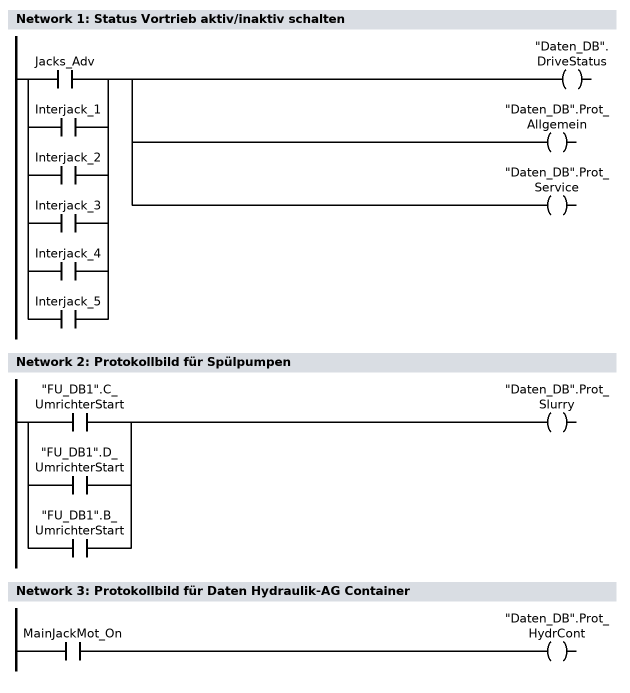
NETWORK
TITLE = Status Vortrieb aktiv/inaktiv schalten
      O     "Jacks_Adv";
      O     "Interjack_1";
      O     "Interjack_2";
      O     "Interjack_3";
      O     "Interjack_4";
      O     "Interjack_5";
      =     "Daten_DB".DriveStatus;
      =     "Daten_DB".Prot_Allgemein;
      =     "Daten_DB".Prot_Service;
NETWORK
TITLE = Protokollbild für Spülpumpen
      O     "FU_DB1".C_UmrichterStart;
      O     "FU_DB1".D_UmrichterStart;
      O     "FU_DB1".B_UmrichterStart;
      =     "Daten_DB".Prot_Slurry;
NETWORK
TITLE = Protokollbild für Daten Hydraulik-AG Container
      A     "MainJackMot_On";
      =     "Daten_DB".Prot_HydrCont;
END_FUNCTION

FUNCTION "DP Ausfall" : VOID	// FC 76
TITLE = Auswertung der Slave-Diagnose
AUTHOR : Simdon
FAMILY : Check
NAME : DP_Fail
VERSION : 0.1
BEGIN
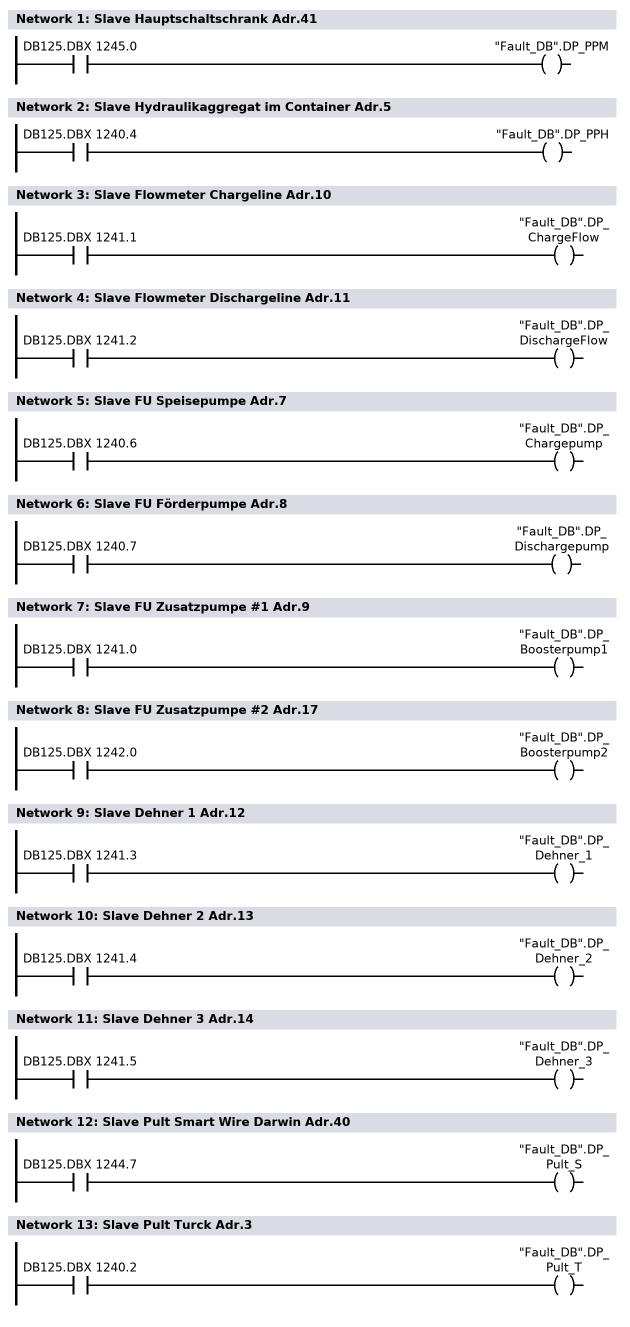
NETWORK
TITLE = Slave Hauptschaltschrank Adr.41
      A     DB125.DBX 1245.0;
      =     "Fault_DB".DP_PPM;
NETWORK
TITLE = Slave Hydraulikaggregat im Container Adr.5
      A     DB125.DBX 1240.4;
      =     "Fault_DB".DP_PPH;
NETWORK
TITLE = Slave Flowmeter Chargeline Adr.10
      A     DB125.DBX 1241.1;
      =     "Fault_DB".DP_ChargeFlow;
NETWORK
TITLE = Slave Flowmeter Dischargeline Adr.11
      A     DB125.DBX 1241.2;
      =     "Fault_DB".DP_DischargeFlow;
NETWORK
TITLE = Slave FU Speisepumpe Adr.7
      A     DB125.DBX 1240.6;
      =     "Fault_DB".DP_Chargepump;
NETWORK
TITLE = Slave FU Förderpumpe Adr.8
      A     DB125.DBX 1240.7;
      =     "Fault_DB".DP_Dischargepump;
NETWORK
TITLE = Slave FU Zusatzpumpe #1 Adr.9
      A     DB125.DBX 1241.0;
      =     "Fault_DB".DP_Boosterpump1;
NETWORK
TITLE = Slave FU Zusatzpumpe #2 Adr.17
      A     DB125.DBX 1242.0;
      =     "Fault_DB".DP_Boosterpump2;
NETWORK
TITLE = Slave Dehner 1 Adr.12
      A     DB125.DBX 1241.3;
      =     "Fault_DB".DP_Dehner_1;
NETWORK
TITLE = Slave Dehner 2 Adr.13
      A     DB125.DBX 1241.4;
      =     "Fault_DB".DP_Dehner_2;
NETWORK
TITLE = Slave Dehner 3 Adr.14
      A     DB125.DBX 1241.5;
      =     "Fault_DB".DP_Dehner_3;
NETWORK
TITLE = Slave Pult Smart Wire Darwin Adr.40
      A     DB125.DBX 1244.7;
      =     "Fault_DB".DP_Pult_S;
NETWORK
TITLE = Slave Pult Turck Adr.3
      A     DB125.DBX 1240.2;
      =     "Fault_DB".DP_Pult_T;
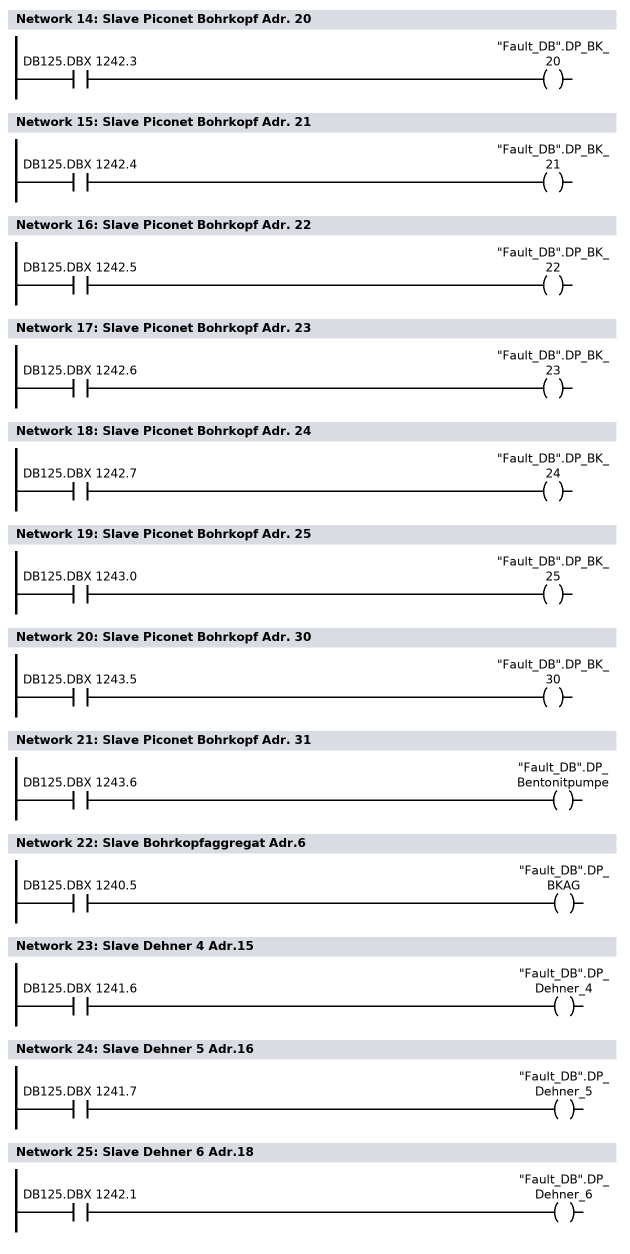
NETWORK
TITLE = Slave Piconet Bohrkopf Adr. 20
      A     DB125.DBX 1242.3;
      =     "Fault_DB".DP_BK_20;
NETWORK
TITLE = Slave Piconet Bohrkopf Adr. 21
      A     DB125.DBX 1242.4;
      =     "Fault_DB".DP_BK_21;
NETWORK
TITLE = Slave Piconet Bohrkopf Adr. 22
      A     DB125.DBX 1242.5;
      =     "Fault_DB".DP_BK_22;
NETWORK
TITLE = Slave Piconet Bohrkopf Adr. 23
      A     DB125.DBX 1242.6;
      =     "Fault_DB".DP_BK_23;
NETWORK
TITLE = Slave Piconet Bohrkopf Adr. 24
      A     DB125.DBX 1242.7;
      =     "Fault_DB".DP_BK_24;
NETWORK
TITLE = Slave Piconet Bohrkopf Adr. 25
      A     DB125.DBX 1243.0;
      =     "Fault_DB".DP_BK_25;
NETWORK
TITLE = Slave Piconet Bohrkopf Adr. 30
      A     DB125.DBX 1243.5;
      =     "Fault_DB".DP_BK_30;
NETWORK
TITLE = Slave Piconet Bohrkopf Adr. 31
      A     DB125.DBX 1243.6;
      =     "Fault_DB".DP_Bentonitpumpe;
NETWORK
TITLE = Slave Bohrkopfaggregat Adr.6
      A     DB125.DBX 1240.5;
      =     "Fault_DB".DP_BKAG;
NETWORK
TITLE = Slave Dehner 4 Adr.15
      A     DB125.DBX 1241.6;
      =     "Fault_DB".DP_Dehner_4;
NETWORK
TITLE = Slave Dehner 5 Adr.16
      A     DB125.DBX 1241.7;
      =     "Fault_DB".DP_Dehner_5;
NETWORK
TITLE = Slave Dehner 6 Adr.18
      A     DB125.DBX 1242.1;
      =     "Fault_DB".DP_Dehner_6;
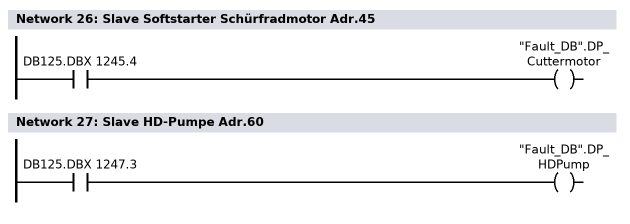
NETWORK
TITLE = Slave Softstarter Schürfradmotor Adr.45
      A     DB125.DBX 1245.4;
      =     "Fault_DB".DP_Cuttermotor;
NETWORK
TITLE = Slave HD-Pumpe Adr.60
      A     DB125.DBX 1247.3;
      =     "Fault_DB".DP_HDPump;
END_FUNCTION

FUNCTION "Sensor_Init" : VOID	// FC 77
TITLE = Sensoren im Bohrkopf initialisieren wenn BK aus
AUTHOR : Simdon
FAMILY : PresBK
NAME : SensBK
VERSION : 0.1
BEGIN
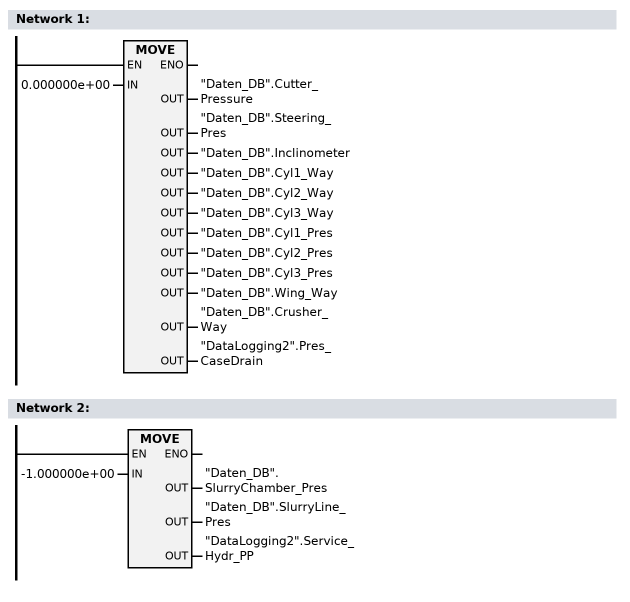
NETWORK
TITLE =
      L     0.000000e+00;
      T     "Daten_DB".Cutter_Pressure;
      T     "Daten_DB".Steering_Pres;
      T     "Daten_DB".Inclinometer;
      T     "Daten_DB".Cyl1_Way;
      T     "Daten_DB".Cyl2_Way;
      T     "Daten_DB".Cyl3_Way;
      T     "Daten_DB".Cyl1_Pres;
      T     "Daten_DB".Cyl2_Pres;
      T     "Daten_DB".Cyl3_Pres;
      T     "Daten_DB".Wing_Way;
      T     "Daten_DB".Crusher_Way;
      T     "DataLogging2".Pres_CaseDrain;
NETWORK
TITLE =
      L     -1.000000e+00;
      T     "Daten_DB".SlurryChamber_Pres;
      T     "Daten_DB".SlurryLine_Pres;
      T     "DataLogging2".Service_Hydr_PP;
END_FUNCTION

FUNCTION "Coolingcircuit_V2" : VOID	// FC 79
TITLE = Kühlkreislauf für den Bohrkopfmotor
AUTHOR : Simdon
FAMILY : Motors
NAME : Cooling
VERSION : 0.1
VAR_TEMP
  P_Cool_Fault : BOOL ;	//Druck Kühlaggregat P<0,6 bar
  P_Diff_Fault : BOOL ;	//Druckdifferenz Eingang/Ausgang Kühlaggregat nicht vorhanden
  P_Diff_Cool : REAL ;	//Druckdifferenz Eingang/Ausgang
END_VAR
BEGIN
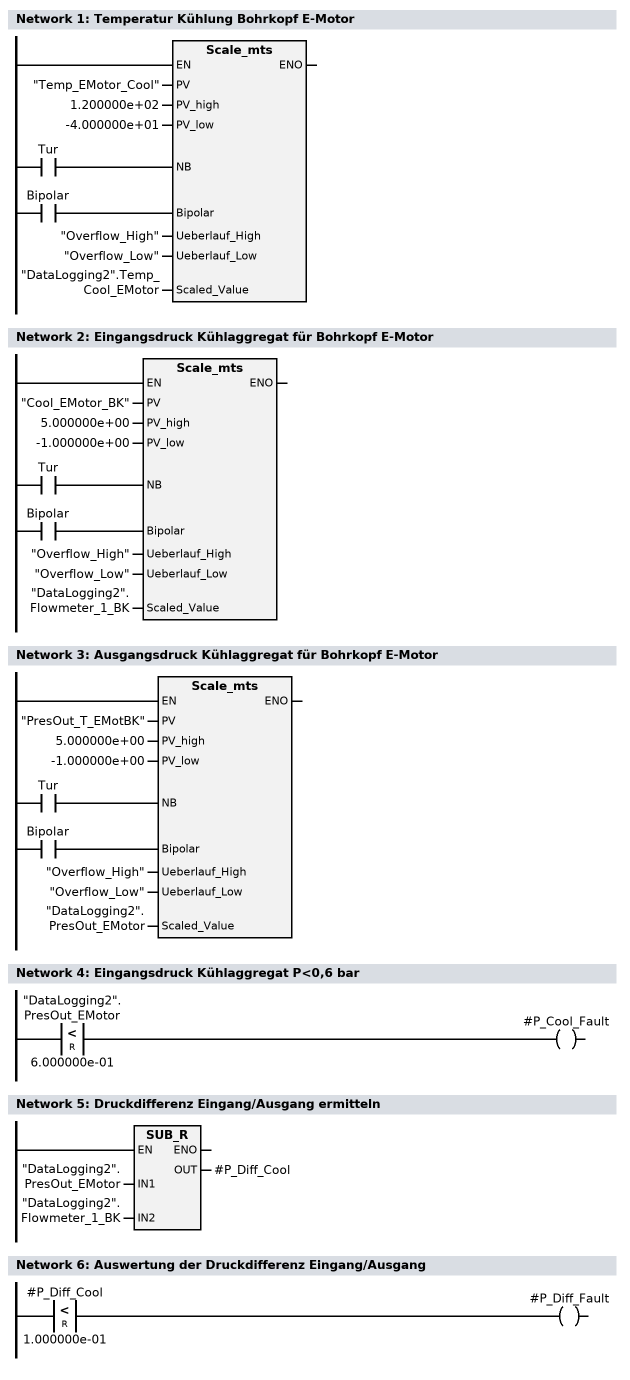
NETWORK
TITLE = Temperatur Kühlung Bohrkopf E-Motor
      A     "Tur";
      =     L 6.0;
      BLD   103;
      A     "Bipolar";
      =     L 6.1;
      BLD   103;
      CALL  "Scale_mts" (
           PV                       := "Temp_EMotor_Cool",
           PV_high                  := 1.200000e+02,
           PV_low                   := -4.000000e+01,
           NB                       := L 6.0,
           Bipolar                  := L 6.1,
           Ueberlauf_High           := "Overflow_High",
           Ueberlauf_Low            := "Overflow_Low",
           Scaled_Value             := "DataLogging2".Temp_Cool_EMotor);
      NOP   0;
NETWORK
TITLE = Eingangsdruck Kühlaggregat für Bohrkopf E-Motor
      A     "Tur";
      =     L 6.0;
      BLD   103;
      A     "Bipolar";
      =     L 6.1;
      BLD   103;
      CALL  "Scale_mts" (
           PV                       := "Cool_EMotor_BK",
           PV_high                  := 5.000000e+00,
           PV_low                   := -1.000000e+00,
           NB                       := L 6.0,
           Bipolar                  := L 6.1,
           Ueberlauf_High           := "Overflow_High",
           Ueberlauf_Low            := "Overflow_Low",
           Scaled_Value             := "DataLogging2".Flowmeter_1_BK);
      NOP   0;
NETWORK
TITLE = Ausgangsdruck Kühlaggregat für Bohrkopf E-Motor
      A     "Tur";
      =     L 6.0;
      BLD   103;
      A     "Bipolar";
      =     L 6.1;
      BLD   103;
      CALL  "Scale_mts" (
           PV                       := "PresOut_T_EMotBK",
           PV_high                  := 5.000000e+00,
           PV_low                   := -1.000000e+00,
           NB                       := L 6.0,
           Bipolar                  := L 6.1,
           Ueberlauf_High           := "Overflow_High",
           Ueberlauf_Low            := "Overflow_Low",
           Scaled_Value             := "DataLogging2".PresOut_EMotor);
      NOP   0;
NETWORK
TITLE = Eingangsdruck Kühlaggregat P<0,6 bar
      L     "DataLogging2".PresOut_EMotor;
      L     6.000000e-01;
      <R;
      =     #P_Cool_Fault;
NETWORK
TITLE = Druckdifferenz Eingang/Ausgang ermitteln
      L     "DataLogging2".PresOut_EMotor;
      L     "DataLogging2".Flowmeter_1_BK;
      -R;
      T     #P_Diff_Cool;
      NOP   0;
NETWORK
TITLE = Auswertung der Druckdifferenz Eingang/Ausgang
      L     #P_Diff_Cool;
      L     1.000000e-01;
      <R;
      =     #P_Diff_Fault;
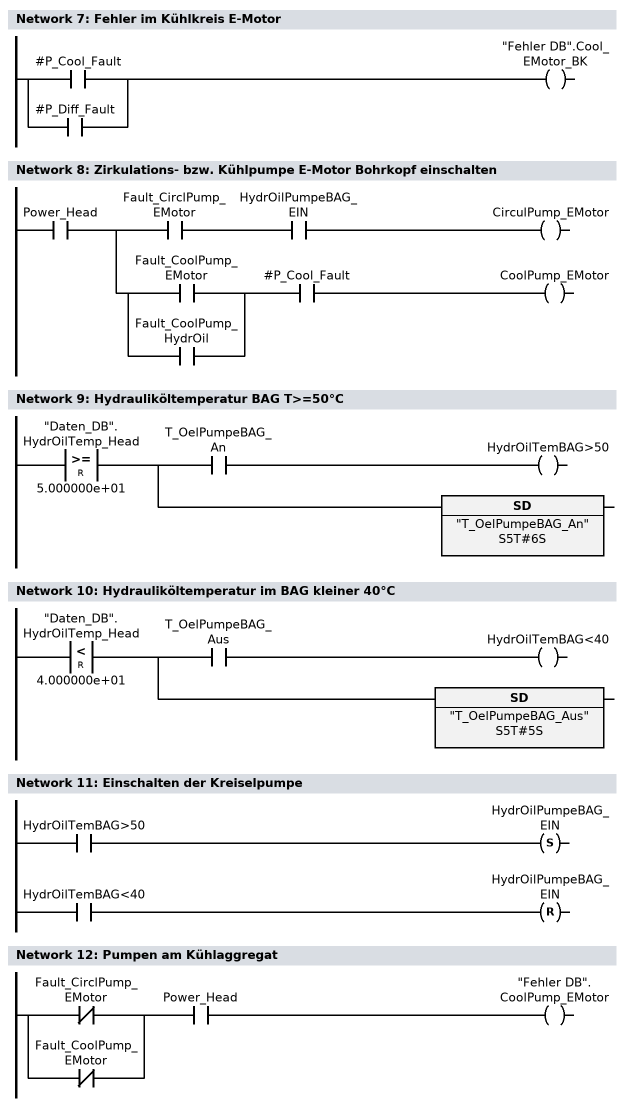
NETWORK
TITLE = Fehler im Kühlkreis E-Motor
      O     #P_Cool_Fault;
      O     #P_Diff_Fault;
      =     "Fehler DB".Cool_EMotor_BK;
NETWORK
TITLE = Zirkulations- bzw. Kühlpumpe E-Motor Bohrkopf einschalten
      A     "Power_Head";
      =     L 6.0;
      A     L 6.0;
      A     "Fault_CirclPump_EMotor";
      A     "HydrOilPumpeBAG_EIN";
      =     "CirculPump_EMotor";
      A     L 6.0;
      A(;
      O     "Fault_CoolPump_EMotor";
      O     "Fault_CoolPump_HydrOil";
      );
      A     #P_Cool_Fault;
      =     "CoolPump_EMotor";
NETWORK
TITLE = Hydrauliköltemperatur BAG T>=50°C
      L     "Daten_DB".HydrOilTemp_Head;
      L     5.000000e+01;
      >=R;
      =     L 6.0;
      A     L 6.0;
      A     "T_OelPumpeBAG_An";
      =     "HydrOilTemBAG>50";
      A     L 6.0;
      BLD   102;
      L     S5T#6S;
      SD    "T_OelPumpeBAG_An";
NETWORK
TITLE = Hydrauliköltemperatur im BAG kleiner 40°C
      L     "Daten_DB".HydrOilTemp_Head;
      L     4.000000e+01;
      <R;
      =     L 6.0;
      A     L 6.0;
      A     "T_OelPumpeBAG_Aus";
      =     "HydrOilTemBAG<40";
      A     L 6.0;
      BLD   102;
      L     S5T#5S;
      SD    "T_OelPumpeBAG_Aus";
NETWORK
TITLE = Einschalten der Kreiselpumpe
      A     "HydrOilTemBAG>50";
      S     "HydrOilPumpeBAG_EIN";
      A     "HydrOilTemBAG<40";
      R     "HydrOilPumpeBAG_EIN";
      NOP   0;
NETWORK
TITLE = Pumpen am Kühlaggregat
      A(;
      ON    "Fault_CirclPump_EMotor";
      ON    "Fault_CoolPump_EMotor";
      );
      A     "Power_Head";
      =     "Fehler DB".CoolPump_EMotor;
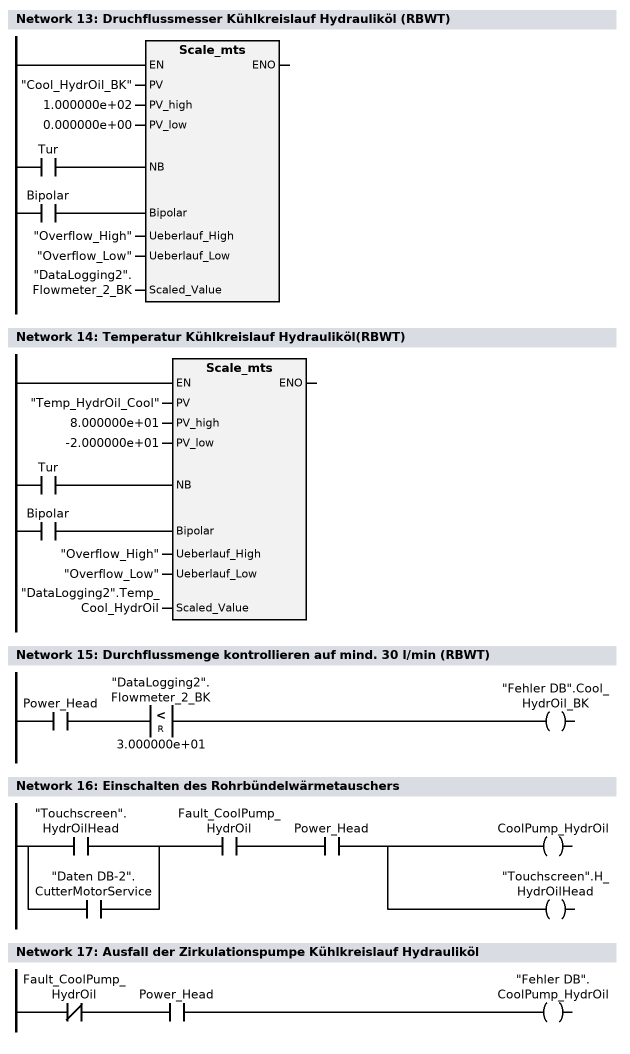
NETWORK
TITLE = Druchflussmesser Kühlkreislauf Hydrauliköl (RBWT)
      A     "Tur";
      =     L 6.0;
      BLD   103;
      A     "Bipolar";
      =     L 6.1;
      BLD   103;
      CALL  "Scale_mts" (
           PV                       := "Cool_HydrOil_BK",
           PV_high                  := 1.000000e+02,
           PV_low                   := 0.000000e+00,
           NB                       := L 6.0,
           Bipolar                  := L 6.1,
           Ueberlauf_High           := "Overflow_High",
           Ueberlauf_Low            := "Overflow_Low",
           Scaled_Value             := "DataLogging2".Flowmeter_2_BK);
      NOP   0;
NETWORK
TITLE = Temperatur Kühlkreislauf Hydrauliköl(RBWT)
      A     "Tur";
      =     L 6.0;
      BLD   103;
      A     "Bipolar";
      =     L 6.1;
      BLD   103;
      CALL  "Scale_mts" (
           PV                       := "Temp_HydrOil_Cool",
           PV_high                  := 8.000000e+01,
           PV_low                   := -2.000000e+01,
           NB                       := L 6.0,
           Bipolar                  := L 6.1,
           Ueberlauf_High           := "Overflow_High",
           Ueberlauf_Low            := "Overflow_Low",
           Scaled_Value             := "DataLogging2".Temp_Cool_HydrOil);
      NOP   0;
NETWORK
TITLE = Durchflussmenge kontrollieren auf mind. 30 l/min (RBWT)
      A     "Power_Head";
      A(;
      L     "DataLogging2".Flowmeter_2_BK;
      L     3.000000e+01;
      <R;
      );
      =     "Fehler DB".Cool_HydrOil_BK;
NETWORK
TITLE = Einschalten des Rohrbündelwärmetauschers
      A(;
      O     "Touchscreen".HydrOilHead;
      O     "Daten DB-2".CutterMotorService;
      );
      A     "Fault_CoolPump_HydrOil";
      A     "Power_Head";
      =     "CoolPump_HydrOil";
      =     "Touchscreen".H_HydrOilHead;
NETWORK
TITLE = Ausfall der Zirkulationspumpe Kühlkreislauf Hydrauliköl
      AN    "Fault_CoolPump_HydrOil";
      A     "Power_Head";
      =     "Fehler DB".CoolPump_HydrOil;
END_FUNCTION

FUNCTION "TACS" : VOID	// FC 80
TITLE = TACS Target
AUTHOR : Simdon
FAMILY : Head
NAME : TACS
VERSION : 0.1
VAR_TEMP
  TargetInfo : INT ;	//Statusmeldung der TACS-Zieltafel
  No_SingleFault : BOOL ;	//Sprung wenn Sammelfehler
  Inclino_ist : REAL ;
END_VAR
BEGIN
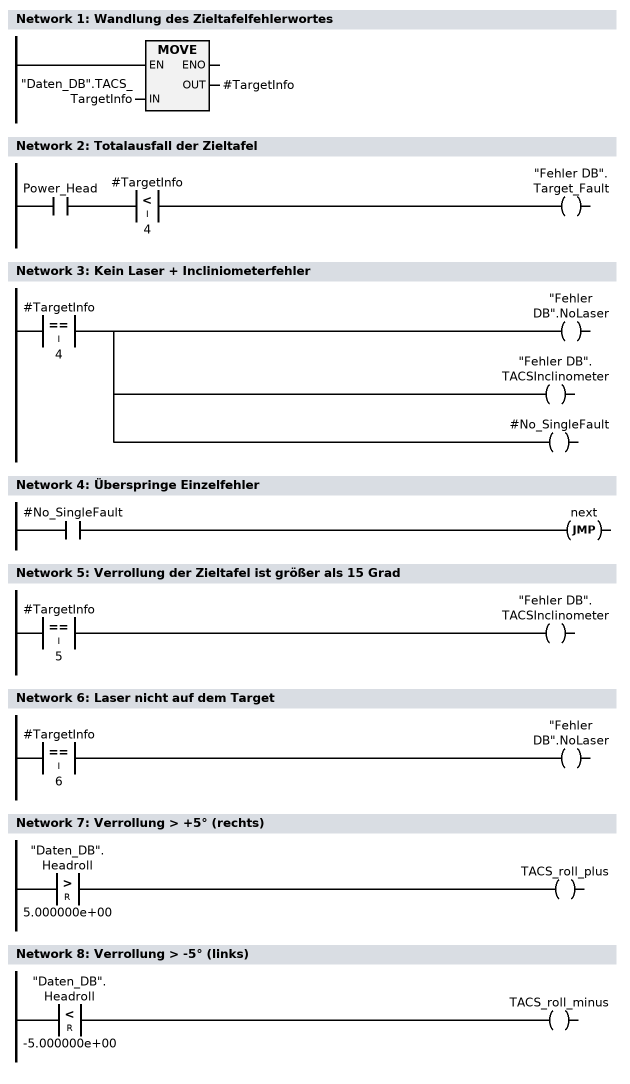
NETWORK
TITLE = Wandlung des Zieltafelfehlerwortes
      L     "Daten_DB".TACS_TargetInfo;
      T     #TargetInfo;
      NOP   0;
NETWORK
TITLE = Totalausfall der Zieltafel
      A     "Power_Head";
      A(;
      L     #TargetInfo;
      L     4;
      <I;
      );
      =     "Fehler DB".Target_Fault;
NETWORK
TITLE = Kein Laser + Incliniometerfehler
      L     #TargetInfo;
      L     4;
      ==I;
      =     "Fehler DB".NoLaser;
      =     "Fehler DB".TACSInclinometer;
      =     #No_SingleFault;
NETWORK
TITLE = Überspringe Einzelfehler
      A     #No_SingleFault;
      JC    next;
NETWORK
TITLE = Verrollung der Zieltafel ist größer als 15 Grad
      L     #TargetInfo;
      L     5;
      ==I;
      =     "Fehler DB".TACSInclinometer;
NETWORK
TITLE = Laser nicht auf dem Target
      L     #TargetInfo;
      L     6;
      ==I;
      =     "Fehler DB".NoLaser;
NETWORK
TITLE = Verrollung > +5° (rechts)
next: L     "Daten_DB".Headroll;
      L     5.000000e+00;
      >R;
      =     "TACS_roll_plus";
NETWORK
TITLE = Verrollung > -5° (links)
      L     "Daten_DB".Headroll;
      L     -5.000000e+00;
      <R;
      =     "TACS_roll_minus";
END_FUNCTION

FUNCTION "mts Inclinometer" : VOID	// FC 81
TITLE = mts Inclinometer
AUTHOR : Simdon
FAMILY : Head
NAME : Inclino
VERSION : 0.1
VAR_TEMP
  TargetInfo : INT ;	//Statusmeldung der TACS-Zieltafel
  No_SingleFault : BOOL ;	//Sprung wenn Sammelfehler
  Inclino_ist : REAL ;
  InclinoMinus : REAL ;
  Neigung_ist : REAL ;
END_VAR
BEGIN
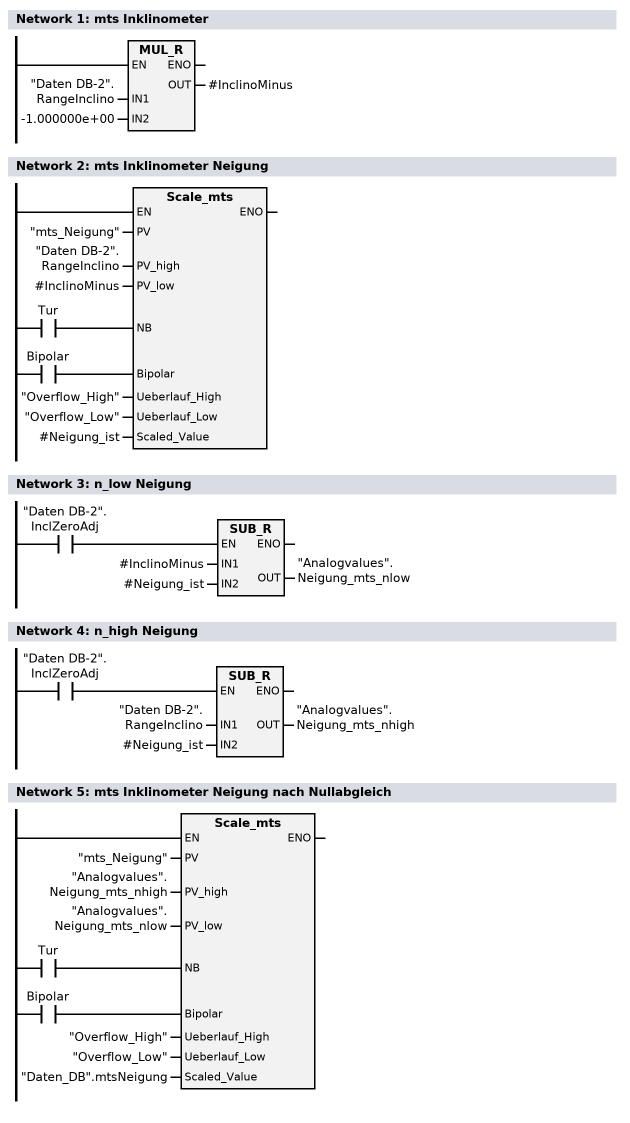
NETWORK
TITLE = mts Inklinometer
      L     "Daten DB-2".RangeInclino;
      L     -1.000000e+00;
      *R;
      T     #InclinoMinus;
      NOP   0;
NETWORK
TITLE = mts Inklinometer Neigung
      A     "Tur";
      =     L 16.0;
      BLD   103;
      A     "Bipolar";
      =     L 16.1;
      BLD   103;
      CALL  "Scale_mts" (
           PV                       := "mts_Neigung",
           PV_high                  := "Daten DB-2".RangeInclino,
           PV_low                   := #InclinoMinus,
           NB                       := L 16.0,
           Bipolar                  := L 16.1,
           Ueberlauf_High           := "Overflow_High",
           Ueberlauf_Low            := "Overflow_Low",
           Scaled_Value             := #Neigung_ist);
      NOP   0;
NETWORK
TITLE = n_low Neigung
//Untergrenze der technischen Einheit nach durchgeführtem Nullabgleich.
      A     "Daten DB-2".InclZeroAdj;
      JNB   _003;
      L     #InclinoMinus;
      L     #Neigung_ist;
      -R;
      T     "Analogvalues".Neigung_mts_nlow;
_003: NOP   0;
NETWORK
TITLE = n_high Neigung
//Obergrenze der technischen Einheit nach durchgeführtem Nullabgleich.
      A     "Daten DB-2".InclZeroAdj;
      JNB   _004;
      L     "Daten DB-2".RangeInclino;
      L     #Neigung_ist;
      -R;
      T     "Analogvalues".Neigung_mts_nhigh;
_004: NOP   0;
NETWORK
TITLE = mts Inklinometer Neigung nach Nullabgleich
      A     "Tur";
      =     L 16.0;
      BLD   103;
      A     "Bipolar";
      =     L 16.1;
      BLD   103;
      CALL  "Scale_mts" (
           PV                       := "mts_Neigung",
           PV_high                  := "Analogvalues".Neigung_mts_nhigh,
           PV_low                   := "Analogvalues".Neigung_mts_nlow,
           NB                       := L 16.0,
           Bipolar                  := L 16.1,
           Ueberlauf_High           := "Overflow_High",
           Ueberlauf_Low            := "Overflow_Low",
           Scaled_Value             := "Daten_DB".mtsNeigung);
      NOP   0;
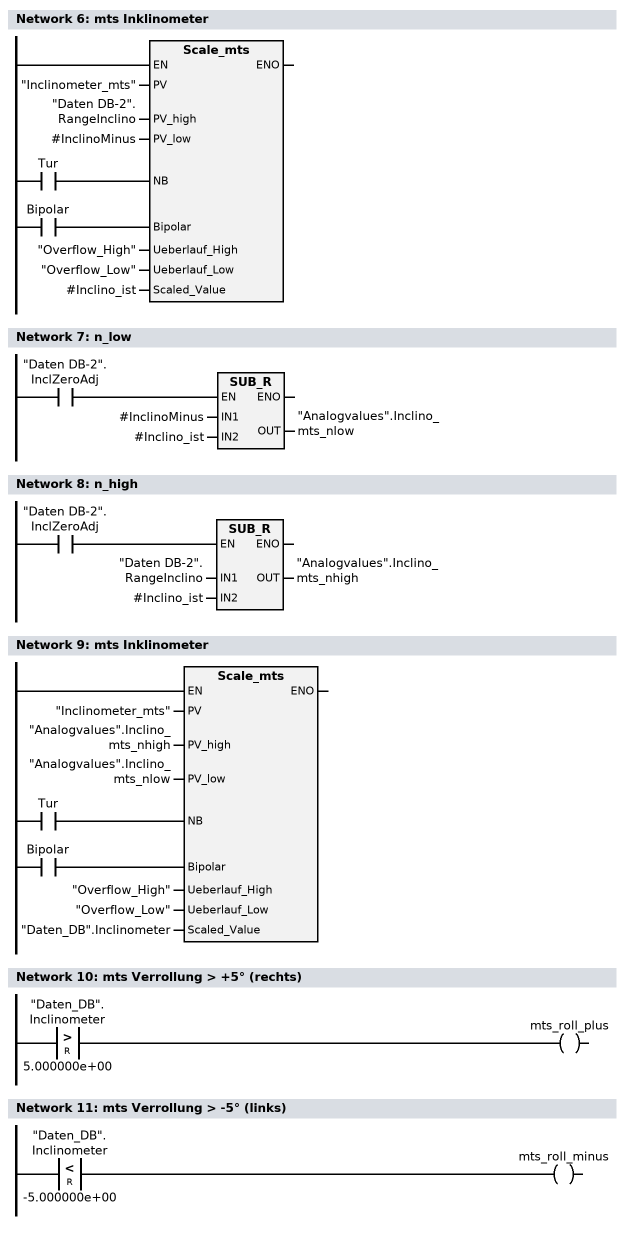
NETWORK
TITLE = mts Inklinometer
      A     "Tur";
      =     L 16.0;
      BLD   103;
      A     "Bipolar";
      =     L 16.1;
      BLD   103;
      CALL  "Scale_mts" (
           PV                       := "Inclinometer_mts",
           PV_high                  := "Daten DB-2".RangeInclino,
           PV_low                   := #InclinoMinus,
           NB                       := L 16.0,
           Bipolar                  := L 16.1,
           Ueberlauf_High           := "Overflow_High",
           Ueberlauf_Low            := "Overflow_Low",
           Scaled_Value             := #Inclino_ist);
      NOP   0;
NETWORK
TITLE = n_low
//Untergrenze der technischen Einheit nach durchgeführtem Nullabgleich.
      A     "Daten DB-2".InclZeroAdj;
      JNB   _005;
      L     #InclinoMinus;
      L     #Inclino_ist;
      -R;
      T     "Analogvalues".Inclino_mts_nlow;
_005: NOP   0;
NETWORK
TITLE = n_high
//Obergrenze der technischen Einheit nach durchgeführtem Nullabgleich.
      A     "Daten DB-2".InclZeroAdj;
      JNB   _006;
      L     "Daten DB-2".RangeInclino;
      L     #Inclino_ist;
      -R;
      T     "Analogvalues".Inclino_mts_nhigh;
_006: NOP   0;
NETWORK
TITLE = mts Inklinometer
      A     "Tur";
      =     L 16.0;
      BLD   103;
      A     "Bipolar";
      =     L 16.1;
      BLD   103;
      CALL  "Scale_mts" (
           PV                       := "Inclinometer_mts",
           PV_high                  := "Analogvalues".Inclino_mts_nhigh,
           PV_low                   := "Analogvalues".Inclino_mts_nlow,
           NB                       := L 16.0,
           Bipolar                  := L 16.1,
           Ueberlauf_High           := "Overflow_High",
           Ueberlauf_Low            := "Overflow_Low",
           Scaled_Value             := "Daten_DB".Inclinometer);
      NOP   0;
NETWORK
TITLE = mts Verrollung > +5° (rechts)
      L     "Daten_DB".Inclinometer;
      L     5.000000e+00;
      >R;
      =     "mts_roll_plus";
NETWORK
TITLE = mts Verrollung > -5° (links)
      L     "Daten_DB".Inclinometer;
      L     -5.000000e+00;
      <R;
      =     "mts_roll_minus";
END_FUNCTION

FUNCTION "Auswertung Verrollung" : VOID	// FC 82
TITLE = Auswertung Verrollung
AUTHOR : Simdon
FAMILY : Head
NAME : Roll
VERSION : 0.1
VAR_TEMP
  C10 : WORD ;
  C11 : INT ;
  C20 : WORD ;
  C21 : INT ;
END_VAR
BEGIN
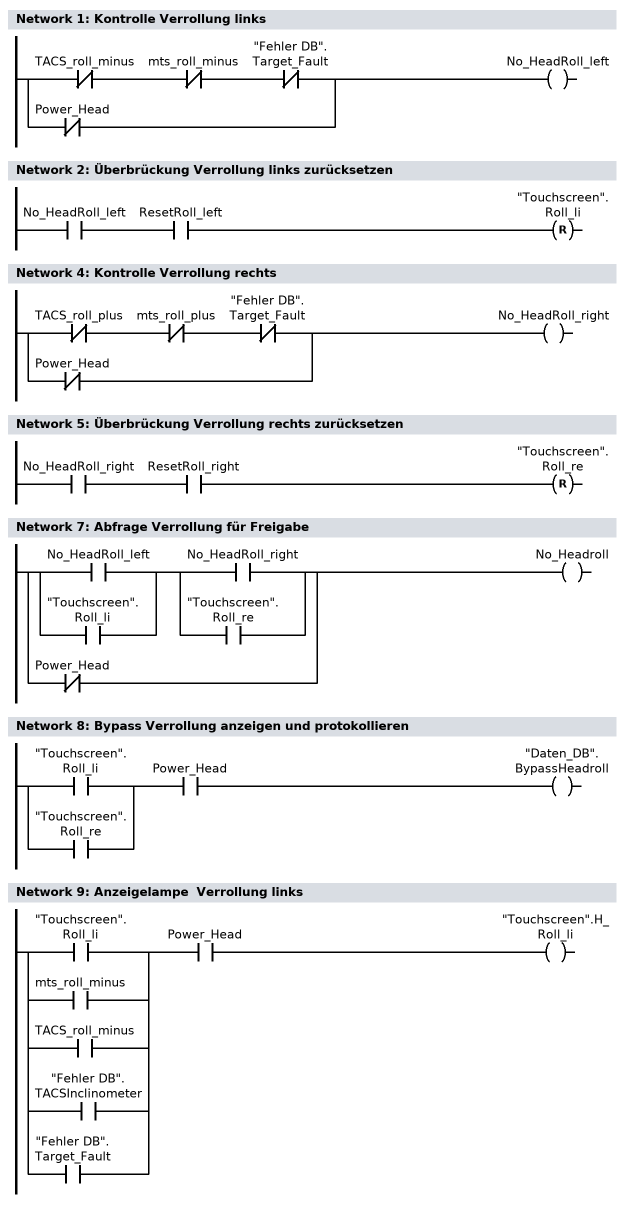
NETWORK
TITLE = Kontrolle Verrollung links
      AN    "TACS_roll_minus";
      AN    "mts_roll_minus";
      AN    "Fehler DB".Target_Fault;
      ON    "Power_Head";
      =     "No_HeadRoll_left";
NETWORK
TITLE = Überbrückung Verrollung links zurücksetzen
      A     "No_HeadRoll_left";
      A     "ResetRoll_left";
      R     "Touchscreen".Roll_li;
NETWORK
TITLE = Verzögerung zum Abschalten der Verrollüberbrückung
      A(;
      A(;
      A     "No_HeadRoll_left";
      A     "Touchscreen".Roll_li;
      A     "Takt_Roll";
      CU    "Z_Roll_Left";
      BLD   101;
      NOP   0;
      NOP   0;
      AN    "Touchscreen".Roll_li;
      R     "Z_Roll_Left";
      NOP   0;
      LC    "Z_Roll_Left";
      T     #C10;
      A     "Z_Roll_Left";
      );
      JNB   _001;
      L     #C10;
      T     #C11;
      SET;
      SAVE;
      CLR;
_001: A     BR;
      );
      A(;
      L     #C11;
      L     3;
      >I;
      );
      =     "ResetRoll_left";
NETWORK
TITLE = Kontrolle Verrollung rechts
      AN    "TACS_roll_plus";
      AN    "mts_roll_plus";
      AN    "Fehler DB".Target_Fault;
      ON    "Power_Head";
      =     "No_HeadRoll_right";
NETWORK
TITLE = Überbrückung Verrollung rechts zurücksetzen
      A     "No_HeadRoll_right";
      A     "ResetRoll_right";
      R     "Touchscreen".Roll_re;
NETWORK
TITLE = Verzögerung zum Abschalten der Verrollüberbrückung
      A(;
      A(;
      A     "No_HeadRoll_right";
      A     "Touchscreen".Roll_re;
      A     "Takt_Roll";
      CU    "Z_Roll_Right";
      BLD   101;
      NOP   0;
      NOP   0;
      AN    "Touchscreen".Roll_re;
      R     "Z_Roll_Right";
      NOP   0;
      LC    "Z_Roll_Right";
      T     #C20;
      A     "Z_Roll_Right";
      );
      JNB   _002;
      L     #C20;
      T     #C21;
      SET;
      SAVE;
      CLR;
_002: A     BR;
      );
      A(;
      L     #C21;
      L     3;
      >I;
      );
      =     "ResetRoll_right";
NETWORK
TITLE = Abfrage Verrollung für Freigabe
      A(;
      O     "No_HeadRoll_left";
      O     "Touchscreen".Roll_li;
      );
      A(;
      O     "No_HeadRoll_right";
      O     "Touchscreen".Roll_re;
      );
      ON    "Power_Head";
      =     "No_Headroll";
NETWORK
TITLE = Bypass Verrollung anzeigen und protokollieren
      A(;
      O     "Touchscreen".Roll_li;
      O     "Touchscreen".Roll_re;
      );
      A     "Power_Head";
      =     "Daten_DB".BypassHeadroll;
NETWORK
TITLE = Anzeigelampe  Verrollung links
      A(;
      O     "Touchscreen".Roll_li;
      O     "mts_roll_minus";
      O     "TACS_roll_minus";
      O     "Fehler DB".TACSInclinometer;
      O     "Fehler DB".Target_Fault;
      );
      A     "Power_Head";
      =     "Touchscreen".H_Roll_li;
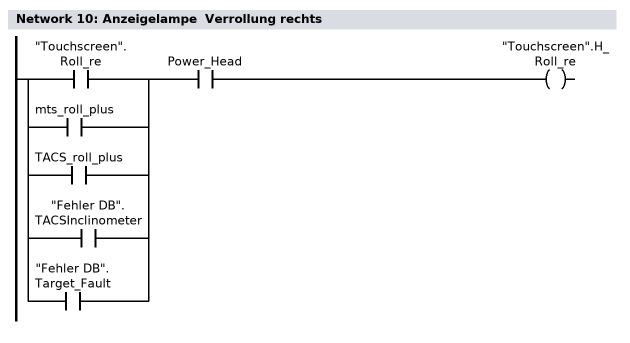
NETWORK
TITLE = Anzeigelampe  Verrollung rechts
      A(;
      O     "Touchscreen".Roll_re;
      O     "mts_roll_plus";
      O     "TACS_roll_plus";
      O     "Fehler DB".TACSInclinometer;
      O     "Fehler DB".Target_Fault;
      );
      A     "Power_Head";
      =     "Touchscreen".H_Roll_re;
END_FUNCTION

FUNCTION "Hochdruck Pumpe" : VOID	// FC 90
TITLE = Ansteuerung der HD-Pumpe über die SPS
AUTHOR : Thiele
FAMILY : Zubehör
NAME : HD-Pumpe
VERSION : 0.1
VAR_TEMP
  HD_Pump : BOOL ;
END_VAR
BEGIN
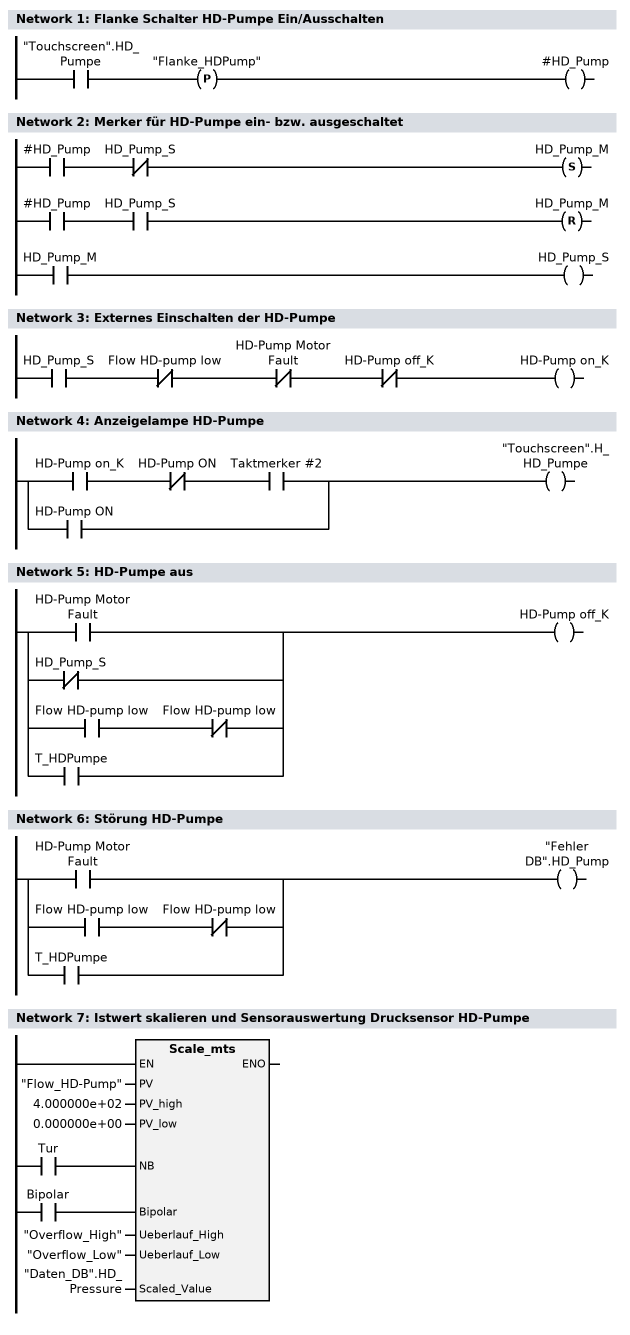
NETWORK
TITLE = Flanke Schalter HD-Pumpe Ein/Ausschalten
      A     "Touchscreen".HD_Pumpe;
      BLD   100;
      FP    "Flanke_HDPump";
      =     #HD_Pump;
NETWORK
TITLE = Merker für HD-Pumpe ein- bzw. ausgeschaltet
      A     #HD_Pump;
      AN    "HD_Pump_S";
      S     "HD_Pump_M";
      A     #HD_Pump;
      A     "HD_Pump_S";
      R     "HD_Pump_M";
      A     "HD_Pump_M";
      =     "HD_Pump_S";
NETWORK
TITLE = Externes Einschalten der HD-Pumpe
      A     "HD_Pump_S";
      AN    "Flow HD-pump low";
      AN    "HD-Pump Motor Fault";
      AN    "HD-Pump off_K";
      =     "HD-Pump on_K";
NETWORK
TITLE = Anzeigelampe HD-Pumpe
      A     "HD-Pump on_K";
      AN    "HD-Pump ON";
      A     "Taktmerker #2";
      O     "HD-Pump ON";
      =     "Touchscreen".H_HD_Pumpe;
NETWORK
TITLE = HD-Pumpe aus
      O     "HD-Pump Motor Fault";
      ON    "HD_Pump_S";
      O;
      A     "Flow HD-pump low";
      AN    "Flow HD-pump low";
      O     "T_HDPumpe";
      =     "HD-Pump off_K";
NETWORK
TITLE = Störung HD-Pumpe
      O     "HD-Pump Motor Fault";
      O;
      A     "Flow HD-pump low";
      AN    "Flow HD-pump low";
      O     "T_HDPumpe";
      =     "Fehler DB".HD_Pump;
NETWORK
TITLE = Istwert skalieren und Sensorauswertung Drucksensor HD-Pumpe
//Istwert des Wegaufnehmers einlesen um die neue Unter- bzw. Obergrenze zur
//Bestimmung des Weges nach dem Nullabgleich. Die Wegaufnehmer liefern ein
//Signal von 4..20 mA.
      A     "Tur";
      =     L 1.0;
      BLD   103;
      A     "Bipolar";
      =     L 1.1;
      BLD   103;
      CALL  "Scale_mts" (
           PV                       := "Flow_HD-Pump",
           PV_high                  := 4.000000e+02,
           PV_low                   := 0.000000e+00,
           NB                       := L 1.0,
           Bipolar                  := L 1.1,
           Ueberlauf_High           := "Overflow_High",
           Ueberlauf_Low            := "Overflow_Low",
           Scaled_Value             := "Daten_DB".HD_Pressure);
      NOP   0;
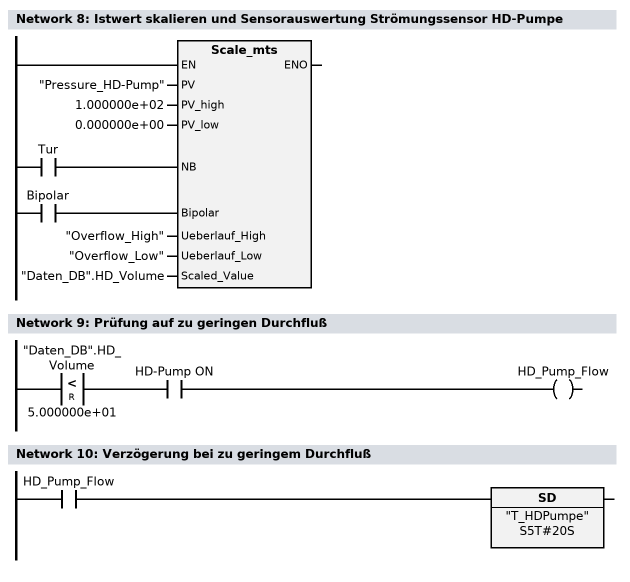
NETWORK
TITLE = Istwert skalieren und Sensorauswertung Strömungssensor HD-Pumpe
//Istwert des Wegaufnehmers einlesen um die neue Unter- bzw. Obergrenze zur
//Bestimmung des Weges nach dem Nullabgleich. Die Wegaufnehmer liefern ein
//Signal von 4..20 mA.
      A     "Tur";
      =     L 1.0;
      BLD   103;
      A     "Bipolar";
      =     L 1.1;
      BLD   103;
      CALL  "Scale_mts" (
           PV                       := "Pressure_HD-Pump",
           PV_high                  := 1.000000e+02,
           PV_low                   := 0.000000e+00,
           NB                       := L 1.0,
           Bipolar                  := L 1.1,
           Ueberlauf_High           := "Overflow_High",
           Ueberlauf_Low            := "Overflow_Low",
           Scaled_Value             := "Daten_DB".HD_Volume);
      NOP   0;
NETWORK
TITLE = Prüfung auf zu geringen Durchfluß
      A(;
      L     "Daten_DB".HD_Volume;
      L     5.000000e+01;
      <R;
      );
      A     "HD-Pump ON";
      =     "HD_Pump_Flow";
NETWORK
TITLE = Verzögerung bei zu geringem Durchfluß
      A     "HD_Pump_Flow";
      L     S5T#20S;
      SD    "T_HDPumpe";
END_FUNCTION

FUNCTION "HD-Valve" : VOID	// FC 91
TITLE = Steuerung der HD-Wasserventile im Bohrkopf
VERSION : 0.1
VAR_TEMP
  temp1 : TIME ;
  temp2 : S5TIME ;
  zahl1 : DINT ;
  zahl2 : DINT ;
  zahl3 : DINT ;
  Set_Valve : BOOL ;	//Zwangsweise ein Ventil einschalten
END_VAR
BEGIN
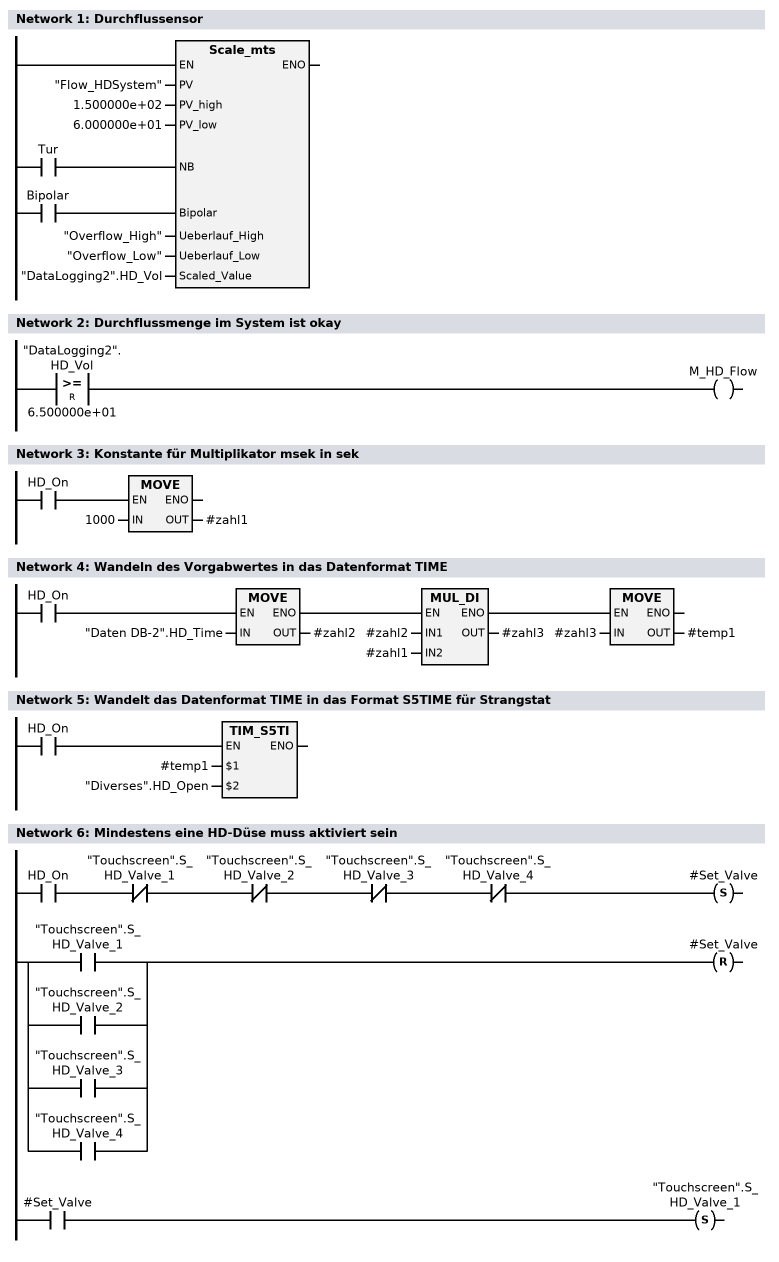
NETWORK
TITLE = Durchflussensor
      A     "Tur";
      =     L 19.0;
      BLD   103;
      A     "Bipolar";
      =     L 19.1;
      BLD   103;
      CALL  "Scale_mts" (
           PV                       := "Flow_HDSystem",
           PV_high                  := 1.500000e+02,
           PV_low                   := 6.000000e+01,
           NB                       := L 19.0,
           Bipolar                  := L 19.1,
           Ueberlauf_High           := "Overflow_High",
           Ueberlauf_Low            := "Overflow_Low",
           Scaled_Value             := "DataLogging2".HD_Vol);
      NOP   0;
NETWORK
TITLE = Durchflussmenge im System ist okay
      L     "DataLogging2".HD_Vol;
      L     6.500000e+01;
      >=R;
      =     "M_HD_Flow";
NETWORK
TITLE = Konstante für Multiplikator msek in sek
      A     "HD_On";
      JNB   _001;
      L     1000;
      T     #zahl1;
_001: NOP   0;
NETWORK
TITLE = Wandeln des Vorgabwertes in das Datenformat TIME
      A(;
      A(;
      A     "HD_On";
      JNB   _004;
      L     "Daten DB-2".HD_Time;
      T     #zahl2;
      SET;
      SAVE;
      CLR;
_004: A     BR;
      );
      JNB   _005;
      L     #zahl2;
      L     #zahl1;
      *D;
      T     #zahl3;
      AN    OV;
      SAVE;
      CLR;
_005: A     BR;
      );
      JNB   _006;
      L     #zahl3;
      T     #temp1;
_006: NOP   0;
NETWORK
TITLE = Wandelt das Datenformat TIME in das Format S5TIME für Strangstat
      A     "HD_On";
      JNB   _007;
      CALL  "TIM_S5TI" (
           $1                       := #temp1,
           $2                       := "Diverses".HD_Open);
_007: NOP   0;
NETWORK
TITLE = Mindestens eine HD-Düse muss aktiviert sein
      A     "HD_On";
      AN    "Touchscreen".S_HD_Valve_1;
      AN    "Touchscreen".S_HD_Valve_2;
      AN    "Touchscreen".S_HD_Valve_3;
      AN    "Touchscreen".S_HD_Valve_4;
      S     #Set_Valve;
      A(;
      O     "Touchscreen".S_HD_Valve_1;
      O     "Touchscreen".S_HD_Valve_2;
      O     "Touchscreen".S_HD_Valve_3;
      O     "Touchscreen".S_HD_Valve_4;
      );
      R     #Set_Valve;
      A     #Set_Valve;
      S     "Touchscreen".S_HD_Valve_1;
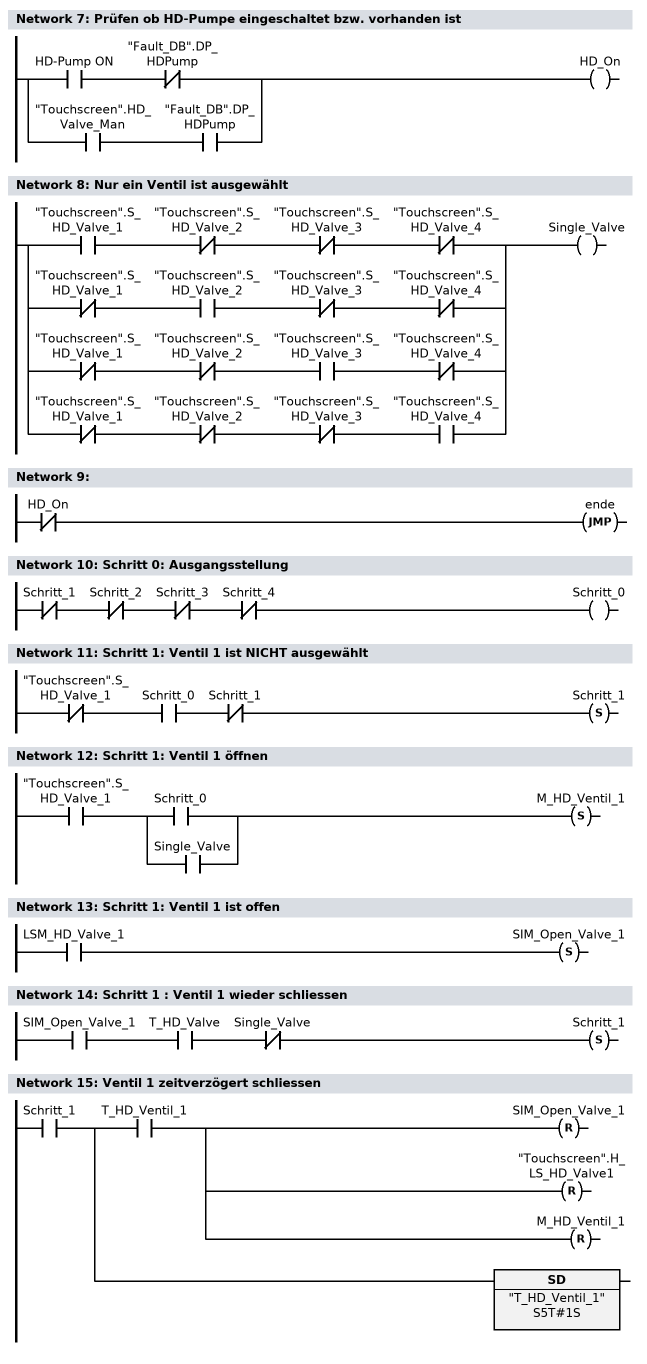
NETWORK
TITLE = Prüfen ob HD-Pumpe eingeschaltet bzw. vorhanden ist
      A     "HD-Pump ON";
      AN    "Fault_DB".DP_HDPump;
      O;
      A     "Touchscreen".HD_Valve_Man;
      A     "Fault_DB".DP_HDPump;
      =     "HD_On";
NETWORK
TITLE = Nur ein Ventil ist ausgewählt
      A     "Touchscreen".S_HD_Valve_1;
      AN    "Touchscreen".S_HD_Valve_2;
      AN    "Touchscreen".S_HD_Valve_3;
      AN    "Touchscreen".S_HD_Valve_4;
      O;
      AN    "Touchscreen".S_HD_Valve_1;
      A     "Touchscreen".S_HD_Valve_2;
      AN    "Touchscreen".S_HD_Valve_3;
      AN    "Touchscreen".S_HD_Valve_4;
      O;
      AN    "Touchscreen".S_HD_Valve_1;
      AN    "Touchscreen".S_HD_Valve_2;
      A     "Touchscreen".S_HD_Valve_3;
      AN    "Touchscreen".S_HD_Valve_4;
      O;
      AN    "Touchscreen".S_HD_Valve_1;
      AN    "Touchscreen".S_HD_Valve_2;
      AN    "Touchscreen".S_HD_Valve_3;
      A     "Touchscreen".S_HD_Valve_4;
      =     "Single_Valve";
NETWORK
TITLE =
      AN    "HD_On";
      JC    ende;
NETWORK
TITLE = Schritt 0: Ausgangsstellung
      AN    "Schritt_1";
      AN    "Schritt_2";
      AN    "Schritt_3";
      AN    "Schritt_4";
      =     "Schritt_0";
NETWORK
TITLE = Schritt 1: Ventil 1 ist NICHT ausgewählt
      AN    "Touchscreen".S_HD_Valve_1;
      A     "Schritt_0";
      AN    "Schritt_1";
      S     "Schritt_1";
NETWORK
TITLE = Schritt 1: Ventil 1 öffnen
      A     "Touchscreen".S_HD_Valve_1;
      A(;
      O     "Schritt_0";
      O     "Single_Valve";
      );
      S     "M_HD_Ventil_1";
NETWORK
TITLE = Schritt 1: Ventil 1 ist offen
      A     "LSM_HD_Valve_1";
      S     "SIM_Open_Valve_1";
NETWORK
TITLE = Schritt 1 : Ventil 1 wieder schliessen
      A     "SIM_Open_Valve_1";
      A     "T_HD_Valve";
      AN    "Single_Valve";
      S     "Schritt_1";
NETWORK
TITLE = Ventil 1 zeitverzögert schliessen
      A     "Schritt_1";
      =     L 19.0;
      A     L 19.0;
      A     "T_HD_Ventil_1";
      R     "SIM_Open_Valve_1";
      R     "Touchscreen".H_LS_HD_Valve1;
      R     "M_HD_Ventil_1";
      A     L 19.0;
      BLD   102;
      L     S5T#1S;
      SD    "T_HD_Ventil_1";
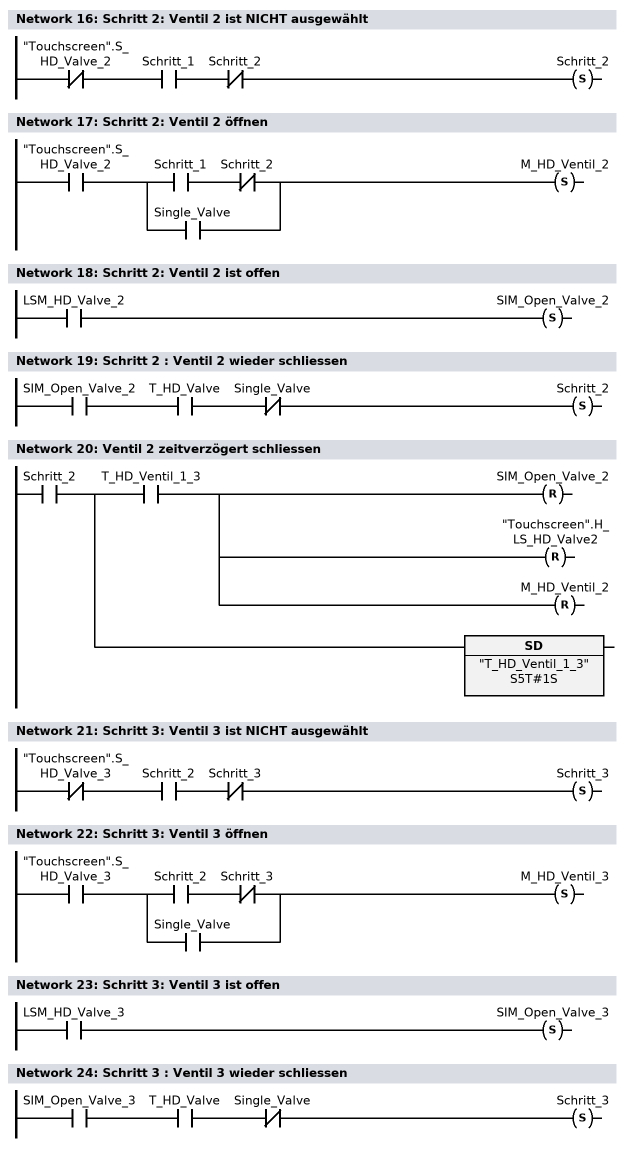
NETWORK
TITLE = Schritt 2: Ventil 2 ist NICHT ausgewählt
      AN    "Touchscreen".S_HD_Valve_2;
      A     "Schritt_1";
      AN    "Schritt_2";
      S     "Schritt_2";
NETWORK
TITLE = Schritt 2: Ventil 2 öffnen
      A     "Touchscreen".S_HD_Valve_2;
      A(;
      A     "Schritt_1";
      AN    "Schritt_2";
      O     "Single_Valve";
      );
      S     "M_HD_Ventil_2";
NETWORK
TITLE = Schritt 2: Ventil 2 ist offen
      A     "LSM_HD_Valve_2";
      S     "SIM_Open_Valve_2";
NETWORK
TITLE = Schritt 2 : Ventil 2 wieder schliessen
      A     "SIM_Open_Valve_2";
      A     "T_HD_Valve";
      AN    "Single_Valve";
      S     "Schritt_2";
NETWORK
TITLE = Ventil 2 zeitverzögert schliessen
      A     "Schritt_2";
      =     L 19.0;
      A     L 19.0;
      A     "T_HD_Ventil_1_3";
      R     "SIM_Open_Valve_2";
      R     "Touchscreen".H_LS_HD_Valve2;
      R     "M_HD_Ventil_2";
      A     L 19.0;
      BLD   102;
      L     S5T#1S;
      SD    "T_HD_Ventil_1_3";
NETWORK
TITLE = Schritt 3: Ventil 3 ist NICHT ausgewählt
      AN    "Touchscreen".S_HD_Valve_3;
      A     "Schritt_2";
      AN    "Schritt_3";
      S     "Schritt_3";
NETWORK
TITLE = Schritt 3: Ventil 3 öffnen
      A     "Touchscreen".S_HD_Valve_3;
      A(;
      A     "Schritt_2";
      AN    "Schritt_3";
      O     "Single_Valve";
      );
      S     "M_HD_Ventil_3";
NETWORK
TITLE = Schritt 3: Ventil 3 ist offen
      A     "LSM_HD_Valve_3";
      S     "SIM_Open_Valve_3";
NETWORK
TITLE = Schritt 3 : Ventil 3 wieder schliessen
      A     "SIM_Open_Valve_3";
      A     "T_HD_Valve";
      AN    "Single_Valve";
      S     "Schritt_3";
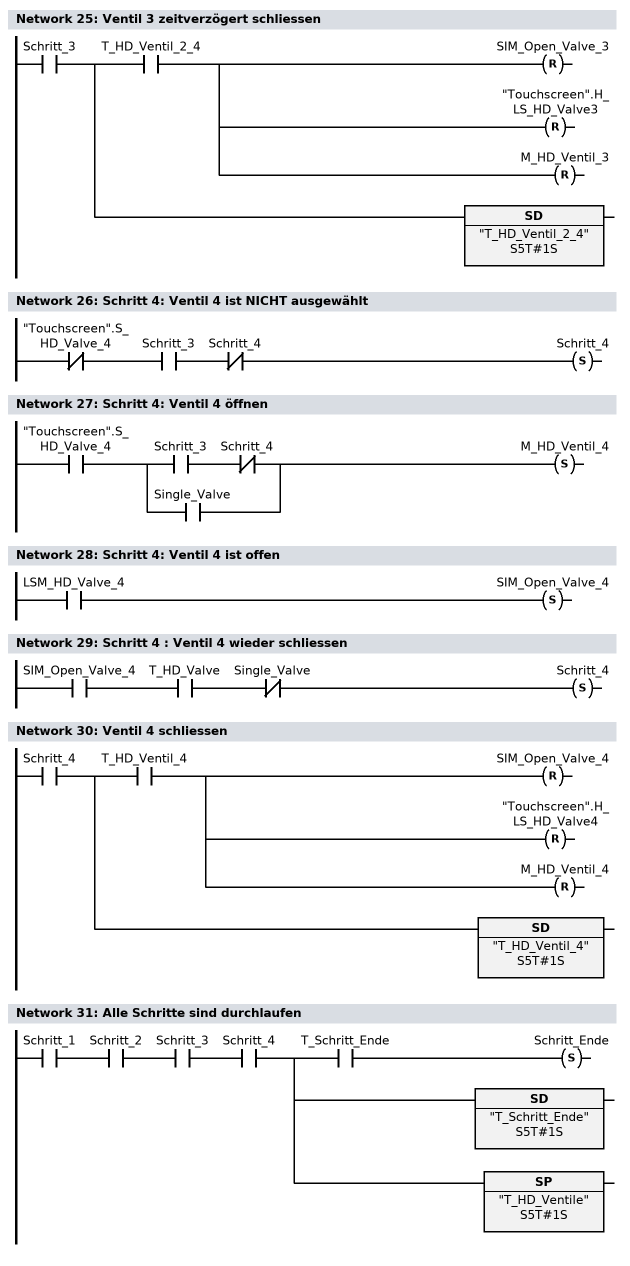
NETWORK
TITLE = Ventil 3 zeitverzögert schliessen
      A     "Schritt_3";
      =     L 19.0;
      A     L 19.0;
      A     "T_HD_Ventil_2_4";
      R     "SIM_Open_Valve_3";
      R     "Touchscreen".H_LS_HD_Valve3;
      R     "M_HD_Ventil_3";
      A     L 19.0;
      BLD   102;
      L     S5T#1S;
      SD    "T_HD_Ventil_2_4";
NETWORK
TITLE = Schritt 4: Ventil 4 ist NICHT ausgewählt
      AN    "Touchscreen".S_HD_Valve_4;
      A     "Schritt_3";
      AN    "Schritt_4";
      S     "Schritt_4";
NETWORK
TITLE = Schritt 4: Ventil 4 öffnen
      A     "Touchscreen".S_HD_Valve_4;
      A(;
      A     "Schritt_3";
      AN    "Schritt_4";
      O     "Single_Valve";
      );
      S     "M_HD_Ventil_4";
NETWORK
TITLE = Schritt 4: Ventil 4 ist offen
      A     "LSM_HD_Valve_4";
      S     "SIM_Open_Valve_4";
NETWORK
TITLE = Schritt 4 : Ventil 4 wieder schliessen
      A     "SIM_Open_Valve_4";
      A     "T_HD_Valve";
      AN    "Single_Valve";
      S     "Schritt_4";
NETWORK
TITLE = Ventil 4 schliessen
      A     "Schritt_4";
      =     L 19.0;
      A     L 19.0;
      A     "T_HD_Ventil_4";
      R     "SIM_Open_Valve_4";
      R     "Touchscreen".H_LS_HD_Valve4;
      R     "M_HD_Ventil_4";
      A     L 19.0;
      BLD   102;
      L     S5T#1S;
      SD    "T_HD_Ventil_4";
NETWORK
TITLE = Alle Schritte sind durchlaufen
      A     "Schritt_1";
      A     "Schritt_2";
      A     "Schritt_3";
      A     "Schritt_4";
      =     L 19.0;
      A     L 19.0;
      A     "T_Schritt_Ende";
      S     "Schritt_Ende";
      A     L 19.0;
      BLD   102;
      L     S5T#1S;
      SD    "T_Schritt_Ende";
      A     L 19.0;
      BLD   102;
      L     S5T#1S;
      SP    "T_HD_Ventile";
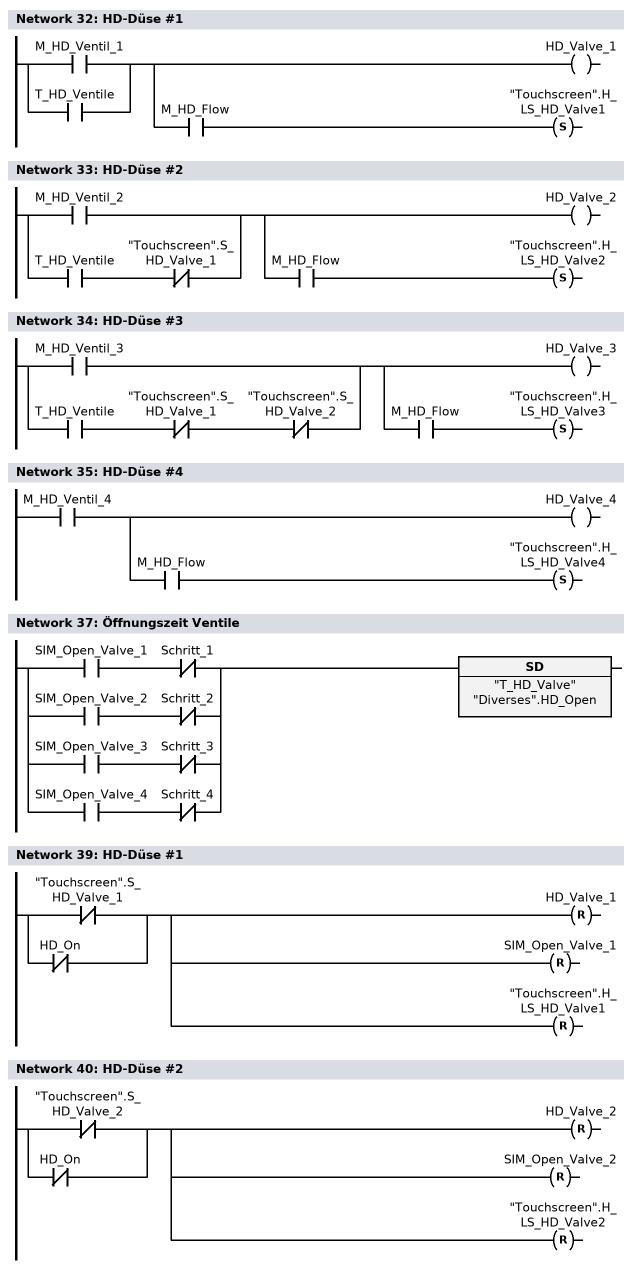
NETWORK
TITLE = HD-Düse #1
      O     "M_HD_Ventil_1";
      O     "T_HD_Ventile";
      =     L 19.0;
      A     L 19.0;
      BLD   102;
      =     "HD_Valve_1";
      A     L 19.0;
      A     "M_HD_Flow";
      S     "Touchscreen".H_LS_HD_Valve1;
NETWORK
TITLE = HD-Düse #2
      O     "M_HD_Ventil_2";
      O;
      A     "T_HD_Ventile";
      AN    "Touchscreen".S_HD_Valve_1;
      =     L 19.0;
      A     L 19.0;
      BLD   102;
      =     "HD_Valve_2";
      A     L 19.0;
      A     "M_HD_Flow";
      S     "Touchscreen".H_LS_HD_Valve2;
NETWORK
TITLE = HD-Düse #3
      O     "M_HD_Ventil_3";
      O;
      A     "T_HD_Ventile";
      AN    "Touchscreen".S_HD_Valve_1;
      AN    "Touchscreen".S_HD_Valve_2;
      =     L 19.0;
      A     L 19.0;
      BLD   102;
      =     "HD_Valve_3";
      A     L 19.0;
      A     "M_HD_Flow";
      S     "Touchscreen".H_LS_HD_Valve3;
NETWORK
TITLE = HD-Düse #4
      A     "M_HD_Ventil_4";
      =     L 19.0;
      A     L 19.0;
      BLD   102;
      =     "HD_Valve_4";
      A     L 19.0;
      A     "M_HD_Flow";
      S     "Touchscreen".H_LS_HD_Valve4;
NETWORK
TITLE = Ende der Schrittkette
      A     "Schritt_Ende";
      JNB   _003;
      CLR;
      =     "Schritt_0";
      =     "Schritt_1";
      =     "Schritt_2";
      =     "Schritt_3";
      =     "Schritt_4";
      =     "Schritt_Ende";
      =     "SIM_Open_Valve_1";
      =     "SIM_Open_Valve_2";
      =     "SIM_Open_Valve_3";
      =     "SIM_Open_Valve_4";
_003: NOP   0;
NETWORK
TITLE = Öffnungszeit Ventile
      A     "SIM_Open_Valve_1";
      AN    "Schritt_1";
      O;
      A     "SIM_Open_Valve_2";
      AN    "Schritt_2";
      O;
      A     "SIM_Open_Valve_3";
      AN    "Schritt_3";
      O;
      A     "SIM_Open_Valve_4";
      AN    "Schritt_4";
      L     "Diverses".HD_Open;
      SD    "T_HD_Valve";
NETWORK
TITLE = HD-Ventile sind ausgeschaltet
ende: AN    "HD_On";
      JNB   _002;
      CLR;
      =     "Schritt_0";
      =     "Schritt_1";
      =     "Schritt_2";
      =     "Schritt_3";
      =     "Schritt_4";
      =     "Schritt_Ende";
      =     "HD_Valve_1";
      =     "HD_Valve_2";
      =     "HD_Valve_3";
      =     "HD_Valve_4";
      =     "M_HD_Ventil_1";
      =     "M_HD_Ventil_2";
      =     "M_HD_Ventil_3";
      =     "M_HD_Ventil_4";
      =     "SIM_Open_Valve_1";
      =     "SIM_Open_Valve_2";
      =     "SIM_Open_Valve_3";
      =     "SIM_Open_Valve_4";
_002: NOP   0;
NETWORK
TITLE = HD-Düse #1
      ON    "Touchscreen".S_HD_Valve_1;
      ON    "HD_On";
      R     "HD_Valve_1";
      R     "SIM_Open_Valve_1";
      R     "Touchscreen".H_LS_HD_Valve1;
NETWORK
TITLE = HD-Düse #2
      ON    "Touchscreen".S_HD_Valve_2;
      ON    "HD_On";
      R     "HD_Valve_2";
      R     "SIM_Open_Valve_2";
      R     "Touchscreen".H_LS_HD_Valve2;
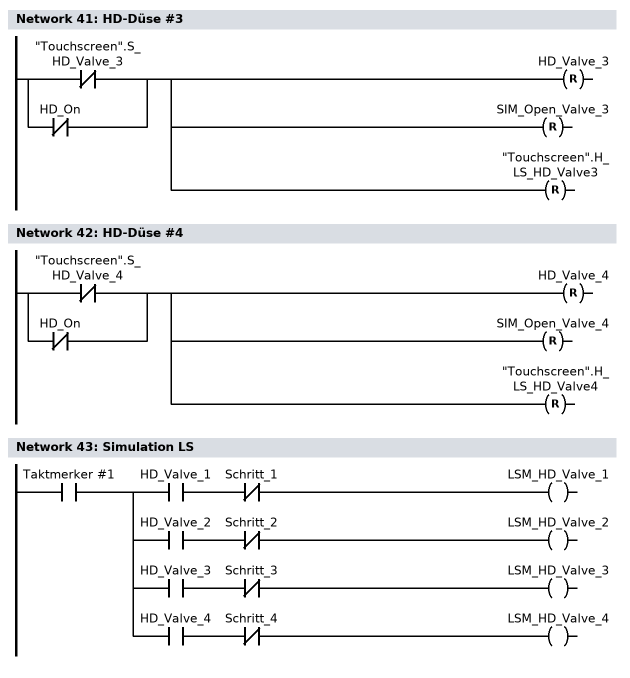
NETWORK
TITLE = HD-Düse #3
      ON    "Touchscreen".S_HD_Valve_3;
      ON    "HD_On";
      R     "HD_Valve_3";
      R     "SIM_Open_Valve_3";
      R     "Touchscreen".H_LS_HD_Valve3;
NETWORK
TITLE = HD-Düse #4
      ON    "Touchscreen".S_HD_Valve_4;
      ON    "HD_On";
      R     "HD_Valve_4";
      R     "SIM_Open_Valve_4";
      R     "Touchscreen".H_LS_HD_Valve4;
NETWORK
TITLE = Simulation LS
      A     "Taktmerker #1";
      =     L 19.0;
      A     L 19.0;
      A     "HD_Valve_1";
      AN    "Schritt_1";
      =     "LSM_HD_Valve_1";
      A     L 19.0;
      A     "HD_Valve_2";
      AN    "Schritt_2";
      =     "LSM_HD_Valve_2";
      A     L 19.0;
      A     "HD_Valve_3";
      AN    "Schritt_3";
      =     "LSM_HD_Valve_3";
      A     L 19.0;
      A     "HD_Valve_4";
      AN    "Schritt_4";
      =     "LSM_HD_Valve_4";
END_FUNCTION

FUNCTION "Cutter Contol mts 2000" : VOID	// FC 95
TITLE = Schürfradsteuerung links/rechts
AUTHOR : Simdon
FAMILY : Cutter
NAME : Cut_Con
VERSION : 0.1
VAR_TEMP
  Mot_okay : BOOL ;	//Antriebsmotor für Hydraulik
  H_Right : BOOL ;
  H_Left : BOOL ;
  Rel_1 : BOOL ;
  Rel_2 : BOOL ;
END_VAR
BEGIN
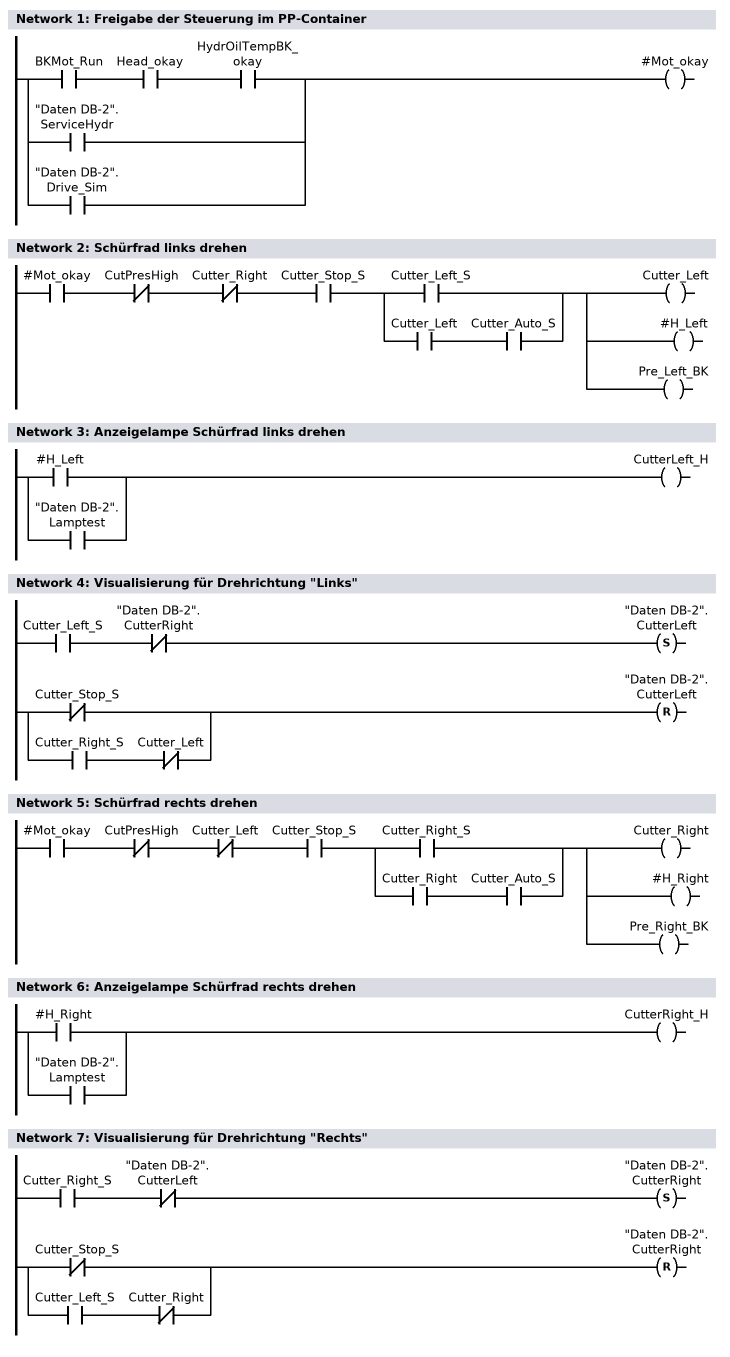
NETWORK
TITLE = Freigabe der Steuerung im PP-Container
      A     "BKMot_Run";
      A     "Head_okay";
      A     "HydrOilTempBK_okay";
      O     "Daten DB-2".ServiceHydr;
      O     "Daten DB-2".Drive_Sim;
      =     #Mot_okay;
NETWORK
TITLE = Schürfrad links drehen
//Schürfrad dreht in einer der gewählten Betriebsarten links herum.
      A     #Mot_okay;
      AN    "CutPresHigh";
      AN    "Cutter_Right";
      A     "Cutter_Stop_S";
      A(;
      O     "Cutter_Left_S";
      O;
      A     "Cutter_Left";
      A     "Cutter_Auto_S";
      );
      =     "Cutter_Left";
      =     #H_Left;
      =     "Pre_Left_BK";
NETWORK
TITLE = Anzeigelampe Schürfrad links drehen
      O     #H_Left;
      O     "Daten DB-2".Lamptest;
      =     "CutterLeft_H";
NETWORK
TITLE = Visualisierung für Drehrichtung "Links"
      A     "Cutter_Left_S";
      AN    "Daten DB-2".CutterRight;
      S     "Daten DB-2".CutterLeft;
      A(;
      ON    "Cutter_Stop_S";
      O;
      A     "Cutter_Right_S";
      AN    "Cutter_Left";
      );
      R     "Daten DB-2".CutterLeft;
      NOP   0;
NETWORK
TITLE = Schürfrad rechts drehen
//Schürfrad dreht in einer der gewählten Betriebsarten rechts herum.
      A     #Mot_okay;
      AN    "CutPresHigh";
      AN    "Cutter_Left";
      A     "Cutter_Stop_S";
      A(;
      O     "Cutter_Right_S";
      O;
      A     "Cutter_Right";
      A     "Cutter_Auto_S";
      );
      =     "Cutter_Right";
      =     #H_Right;
      =     "Pre_Right_BK";
NETWORK
TITLE = Anzeigelampe Schürfrad rechts drehen
      O     #H_Right;
      O     "Daten DB-2".Lamptest;
      =     "CutterRight_H";
NETWORK
TITLE = Visualisierung für Drehrichtung "Rechts"
      A     "Cutter_Right_S";
      AN    "Daten DB-2".CutterLeft;
      S     "Daten DB-2".CutterRight;
      A(;
      ON    "Cutter_Stop_S";
      O;
      A     "Cutter_Left_S";
      AN    "Cutter_Right";
      );
      R     "Daten DB-2".CutterRight;
      NOP   0;
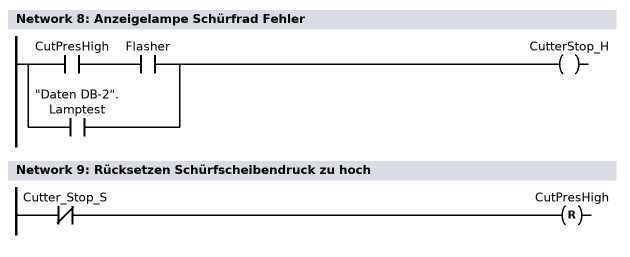
NETWORK
TITLE = Anzeigelampe Schürfrad Fehler
      A     "CutPresHigh";
      A     "Flasher";
      O     "Daten DB-2".Lamptest;
      =     "CutterStop_H";
NETWORK
TITLE = Rücksetzen Schürfscheibendruck zu hoch
      AN    "Cutter_Stop_S";
      R     "CutPresHigh";
END_FUNCTION

FUNCTION "Scale_mts" : VOID	// FC 107
TITLE = Scale Analoginput Uni- und Bipolar
AUTHOR : Simdon
FAMILY : Wandeln
NAME : Scalemts
VERSION : 1.0
VAR_INPUT
  PV : INT ;	//Analogeingabewert (PEW)
  PV_high : REAL ;	//oberer Grenzwert
  PV_low : REAL ;	//unterer Grenzwert
  NB : BOOL ;	//Nennbereich 1=32767, 0=27648
  Bipolar : BOOL ;	//Typ der Baugruppe. 0=Unipolar, 1=Bipolar
END_VAR
VAR_OUTPUT
  Ueberlauf_High : BOOL ;	//Überlauf oberer Bereich
  Ueberlauf_Low : BOOL ;	//Überlauf unterer Bereich
  Scaled_Value : REAL ;	//normierter Analogwert
END_VAR
VAR_TEMP
  PV_Real : REAL ;	//Eingangswert als Real-Zahl
  wb_high : REAL ;	//Obergrenze Wertebereich
  wb_low : REAL ;	//Untergrenze Wertebereich
  ZW_1 : REAL ;	//Zwischenwert
  wb_range : REAL ;	//Wertebereich
  eng_range : REAL ;	//Bereich der tech. Messeinheit
  nb_high : REAL ;	//Nennbereich plus
  nb_low : REAL ;	//Nennbereich minus
END_VAR
BEGIN
NETWORK
TITLE = Nennbereich
//OUT = [ ((IN) – K1)/(K2–K1)) * (HI_LIM–LO_LIM)] + LO_LIM
      A     #NB;	// Prüfen welcher Wertebereich relevant ist
      JC    tur;	// Sprung
      L     2.764800e+04;	// Wertebereich obere Grenze
      T     #nb_high;	// Obere Grenze merken
      L     -2.764800e+04;	// Wertebereich untere Grenze
      T     #nb_low;	// Untere Grenze merken
      JU    go;	// Sprung
tur:  L     3.276700e+04;	// Wertebereich obere Grenze
      T     #nb_high;	// Obere Grenze merken
      L     -3.276800e+04;	// Wertebereich untere Grenze
      T     #nb_low;	// Untere Grenze merken
NETWORK
TITLE = Wandlung von Integer auf Real, Prüfung der Grenzen
//OUT = [ ((IN) – K1)/(K2–K1)) * (HI_LIM–LO_LIM)] + LO_LIM
go:   L     #PV;	// Wert des gemessenen Analogeingangswortes laden
      ITD;	// 16 Bit-Ganzzahl in 32 Bit-Realzahl wandeln
      DTR;	// 32 Bit-Ganzzahl in reelle Zahl speichern
      T     #PV_Real;	// Einganswert als Real merken
      L     #nb_high;	// OberenNennbereich des Analogeinganges
      T     #wb_high;	// Oberen Nennbereich merken
      L     #nb_low;	// Unteren Nennbereich des Analogeinganges bipolar
      A     #Bipolar;	// Prüfung auf Uni- bzw. Bipolaren Eingang
      JC    m001;
      L     0;	// Unteren Nennbereich des Analogeinganges unipolar
m001: T     #wb_low;	// Unteren Nennbereich merken
      L     #PV_Real;	// Einganswert laden
      L     #wb_high;	// Obere Grenze vom Nennbereich laden
      >R;	// Prüfung auf Überlauf
      =     #Ueberlauf_High;	// Auswertung für Überlauf
      L     #PV_Real;	// Einganswert als Real laden
      L     #wb_low;	// Untere Grenze vom Wertebereich laden
      <R;	// Auf Unterlauf prüfen
      =     #Ueberlauf_Low;	// Auswertung auf Unterschreitung
NETWORK
TITLE = Technischer Bereich
      L     #PV_high;	// Istwert-Obergrenze laden
      L     #PV_low;	// Istwert-Untergrenze laden
      -R;	// Obergrenze - Untergrenze
      T     #eng_range;	// Bereich der technischen Maßeinheit speichern
NETWORK
TITLE =
      L     #wb_high;	// Obere Grenze vom Wertebereich laden
      L     #wb_low;	// Untere Grenze vom Wertebereich laden
      -R;	// Wertebereich: Obergrenze - Untergrenze
      T     #wb_range;	// Bereich für Wertebereich speichern
      L     #PV_Real;	// Einganswert als Real laden
      L     #wb_low;	// Untere Grenze vom Wertebereich laden
      -R;	// Einganswert - Unterer Wertebereich
      T     #ZW_1;	// Zwischenwert 1 merken
      L     #wb_range;	// Bereich für Wertebereich  laden
      /R;	// Zwischenwert 1 / Wertebereich
      L     #eng_range;	// Bereich der technischen Maßeinheit laden
      *R;	// Multiplikation
      L     #PV_low;	// Istwert-Untergrenze laden
      +R;	// Addition
      T     #Scaled_Value;	// Endergebnis der Skalierung
END_FUNCTION

FUNCTION "Scale_Poti" : VOID	// FC 108
TITLE = SWD-Poti
AUTHOR : Simdon
FAMILY : Wandeln
NAME : ScalePot
VERSION : 1.0
VAR_INPUT
  Poti : BYTE ;
  Scale_In : INT ;	//Zu skalierender Wert
  Input : REAL ;	//Wertebereich des Eingabewertes
  Offset : INT ;	//Sprung
END_VAR
VAR_OUTPUT
  Scaled_Value : WORD ;	//Skalierter Wert für angesteuertes Gerät
END_VAR
VAR_TEMP
  Ist : INT ;	//Poti zu Integer
  Ist_1 : DINT ;	//Poti zu Double-Integer
  Ist_2 : REAL ;	//Poti zu Real
  Scale_1 : DINT ;	//Steuerwert zu Double-Integer
  Scale_2 : REAL ;	//Steuerwert zu Real
  Zw_1 : REAL ;	//Zwischenberechnung
  Zw_2 : REAL ;	//Zwischenberechnung
  Zw_3 : REAL ;	//Zwischenberechnung
  Zw_4 : DINT ;	//Zwischenberechnung
  Zw_5 : INT ;	//Zwischenberechnung
  Zw_6 : INT ;	//Zwischenberechnung
  Sprung : INT ;
END_VAR
BEGIN
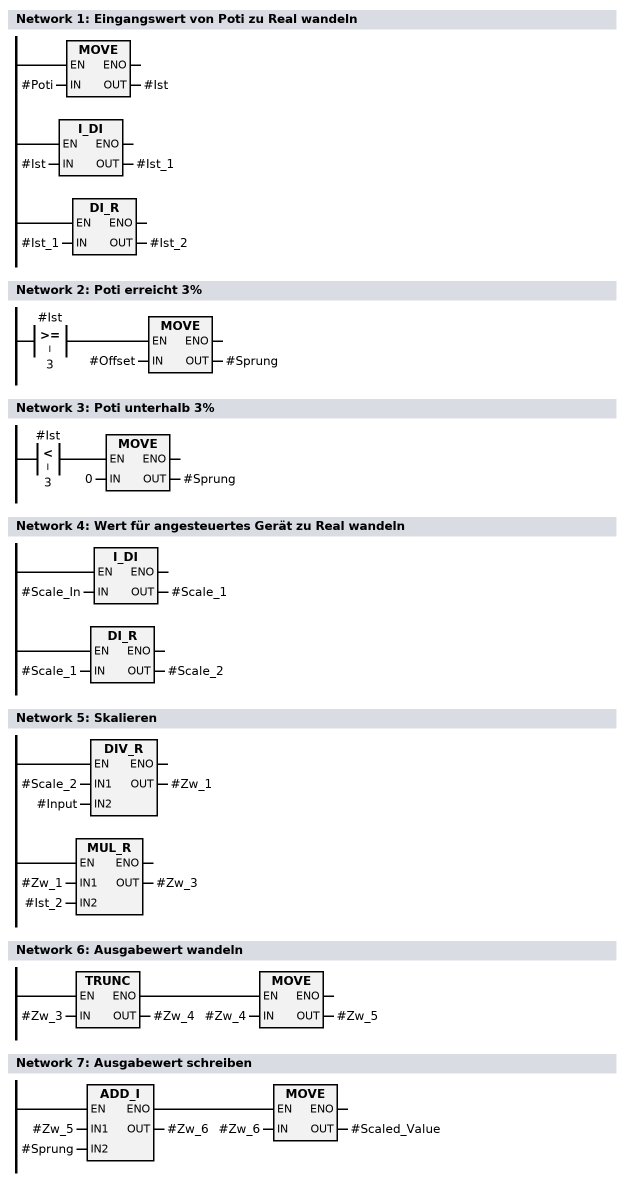
NETWORK
TITLE = Eingangswert von Poti zu Real wandeln
      L     #Poti;
      T     #Ist;
      L     #Ist;
      ITD;
      T     #Ist_1;
      L     #Ist_1;
      DTR;
      T     #Ist_2;
NETWORK
TITLE = Poti erreicht 3%
      A(;
      L     #Ist;
      L     3;
      >=I;
      );
      JNB   _001;
      L     #Offset;
      T     #Sprung;
_001: NOP   0;
NETWORK
TITLE = Poti unterhalb 3%
      A(;
      L     #Ist;
      L     3;
      <I;
      );
      JNB   _002;
      L     0;
      T     #Sprung;
_002: NOP   0;
NETWORK
TITLE = Wert für angesteuertes Gerät zu Real wandeln
      L     #Scale_In;
      ITD;
      T     #Scale_1;
      L     #Scale_1;
      DTR;
      T     #Scale_2;
NETWORK
TITLE = Skalieren
      L     #Scale_2;
      L     #Input;
      /R;
      T     #Zw_1;
      L     #Zw_1;
      L     #Ist_2;
      *R;
      T     #Zw_3;
NETWORK
TITLE = Ausgabewert wandeln
      A(;
      L     #Zw_3;
      TRUNC;
      T     #Zw_4;
      AN    OV;
      SAVE;
      CLR;
      A     BR;
      );
      JNB   _003;
      L     #Zw_4;
      T     #Zw_5;
_003: NOP   0;
NETWORK
TITLE = Ausgabewert schreiben
      A(;
      L     #Zw_5;
      L     #Sprung;
      +I;
      T     #Zw_6;
      AN    OV;
      SAVE;
      CLR;
      A     BR;
      );
      JNB   _004;
      L     #Zw_6;
      T     #Scaled_Value;
_004: NOP   0;
END_FUNCTION

FUNCTION "PKE" : BOOL	// FC 110
TITLE = Motorstarterkombinationen mit PKE
AUTHOR : Simdon
FAMILY : PKE
NAME : PKE-1
VERSION : 0.1
VAR_INPUT
  Daten_DB : INT ;	//Bausteinnummer für Datenablage
  PKE_DB : INT ;	//Bausteinnummer für PKE-Daten
  Offset : INT ;	//Bausteinoffset für Datenablage
  Eingang : INT ;	//Eingangsadresse des PKE (Anfangsadresse)
  IR_Strom : REAL ;	//Maximaler Einstellwert für PKE
END_VAR
VAR_OUTPUT
  RET_VAL : BOOL ;
END_VAR
VAR_TEMP
  Contactor_In : BOOL ;	//Schaltstellung Leistungsschütz
  Status_In : BOOL ;	//Status PKE
  Auto_In : BOOL ;	//Stellung Schalter 1-0-A
  Auto2_In : BOOL ;	//Stellung Schalter 1-0-A
  Failure_In : BOOL ;	//Diagnosemeldung
  Frei1_In : BOOL ;
  Present_In : BOOL ;	//Modul vorhanden
  Frei2_In : BOOL ;
  IR1_In : BOOL ;	//Eingestellter Wert IR
  IR2_In : BOOL ;	//Eingestellter Wert IR
  IR3_In : BOOL ;	//Eingestellter Wert IR
  IR4_In : BOOL ;	//Eingestellter Wert IR
  TRIPR1_In : BOOL ;	//Auslösegrund
  TRIPR2_In : BOOL ;	//Auslösegrund
  TRIPR3_In : BOOL ;	//Auslösegrund
  ACKR_In : BOOL ;	//Acknowledge
  Motorstrom_In : BYTE ;	//Motorstrom
  Therm_In : BYTE ;	//Thermisches Motorabbild
  Block_In : BYTE ;	//Auslöseblock
  IR_1 : WORD ;	//Zwischenwert Auslösestrom
  IR_2 : INT ;	//Zwischenwert Auslösestrom
  TRIPR_1 : WORD ;	//Zwischenwert Auslösegrund
  TRIPR_2 : INT ;	//Zwischenwert Auslösegrund
  IR_Wert : REAL ;	//Gewandelter Wert für Auslösestrom
  IR_High : REAL ;	//Obergrenze für Auslösestrom
  Release : BOOL ;	//Freigabe wenn eingestellter Auslösestrom okay
  iDBNr : INT ;	//Instanz-DB für Datenablage
  Offset2 : INT ;	//Offset für PKE-DB
  EAAdr : DINT ;	//Eingangsadresse für PKE
  RetVal : INT ;
  Block1 : WORD ;	//Zwischenwert für Typ Auslöseblock
  Block2 : INT ;	//Zwischenwert für Typ Auslöseblock
  S_A : BOOL ;	//Stellung 1-0-A-Schalter "A"
  S_0 : BOOL ;	//Stellung 1-0-A-Schalter "0"
  S_1 : BOOL ;	//Stellung 1-0-A-Schalter "1"
  iDB_PKE : INT ;	//Instanz-DB für PKE-Daten
END_VAR
BEGIN
NETWORK
TITLE = Eingangswerte laden und verteilen
      L     #Eingang;	// Anfangsadresse des PKE
      T     #EAAdr;	// Übertragen in temp. Adressmerker
      SLD   3;	// Wort schieben
      LAR1;	// Wert ins Adressregister 1 ablegen
      L     PIB [AR1,P#0.0];	// Eingangsbyte laden
      T     LB 0;	// In Lokaldaten ablegen
      L     PIB [AR1,P#1.0];	// Eingangsbyte laden
      T     LB 1;	// In Lokaldaten ablegen
      L     PIB [AR1,P#2.0];	// Eingangsbyte laden
      T     #Motorstrom_In;	// In Lokaldaten ablegen
      L     PIB [AR1,P#3.0];	// Eingangsbyte laden
      T     #Therm_In;	// In Lokaldaten ablegen
      L     PIB [AR1,P#4.0];	// Eingangsbyte laden
      T     #Block_In;	// In Lokaldaten ablegen
NETWORK
TITLE = Feststellen welcher Auslöseblock eingesetzt wird
      L     #Block_In;	// Kenndaten vom Auslöseblock lesen
      T     #Block1;	// Wandlung zum Wort
      L     W#16#7;	// Typ Auslöseblock maskieren
      AW;
      T     #Block2;	// Als Integer ablegen
      L     #Block2;	// Blocktyp laden
      L     0;	// Vergleich mit PKE 1,2
      ==I;
      JNB   _011;	// Sprung wenn nicht gleich
      L     0;	// Offset für DB zum Datenauslesen
      T     #Offset2;
_011: L     #Block2;	// Blocktyp laden
      L     1;	// Vergleich mit PKE 4
      ==I;
      JNB   _012;	// Sprung wenn nicht gleich
      L     64;	// Offset für DB zum Datenauslesen
      T     #Offset2;	// Offset ablegen
_012: L     #Block2;	// Blocktyp laden
      L     2;	// Vergleich mit PKE 12
      ==I;
      JNB   _013;	// Sprung wenn nicht gleich
      L     128;	// Offset für DB zum Datenauslesen
      T     #Offset2;	// Offset ablegen
_013: L     #Block2;	// Blocktyp laden
      L     3;	// Vergleich mit PKE 32
      ==I;
      JNB   _014;	// Sprung wenn nicht gleich
      L     192;	// Offset für DB zum Datenauslesen
      T     #Offset2;	// Offset ablegen
_014: NOP   0;
NETWORK
TITLE = Eingestellten Wert IR maskieren und wandeln
      L     LB 1;	// Byte 1 vom PKE laden
      T     #IR_1;	// Zwischenspeichern in IR-Werte 1
      L     W#16#F;	// Eingestellten IR-Wert maskieren
      AW;
      T     #IR_2;	// IR-Wert als Integer
NETWORK
TITLE = Auslösegrung TRIPR maskieren und wandeln
//1: Überlastfall; 2: Kurzschluß; 3: Phasenausfall/Phasenunsymetrie
//4: Stellung Test am PKE
      L     LB 1;	// Byte 1 vom PKE laden
      L     #TRIPR_1;	// Zwischenspeichern in TRIPR-Werte 1
      L     W#16#70;	// TRIPR-Wert maskieren
      AW;
      T     #TRIPR_2;	// TRIPR-Wert als Integer
NETWORK
TITLE = Auswertung 1-0-A-Schalter
      A     #Auto_In;	// Stellung 1-0-A-Schalter Bit 1
      AN    #Auto2_In;	// Stellung 1-0-A-Schalter Bit 2
      =     #S_A;	// Schalter in Stellung "A"
      AN    #Auto_In;	// Stellung 1-0-A-Schalter Bit 1
      A     #Auto2_In;	// Stellung 1-0-A-Schalter Bit 2
      =     #S_0;	// Schalter in Stellung "0"
      A     #Auto_In;	// Stellung 1-0-A-Schalter Bit 1
      A     #Auto2_In;	// Stellung 1-0-A-Schalter Bit 2
      =     #S_1;	// Schalter in Stellung "1"
NETWORK
TITLE = DB mit IR Werten für PKE öffnen
      L     #PKE_DB;	// Nummer des DB laden
      T     #iDB_PKE;	// Nummer für Instanz DB übertragen
      OPN   DB [#iDB_PKE];	// Instanz DB öffnen
      LAR2  P#DBX 0.0;	// Pointer auf Anfang
      L     #Offset2;	// Offset für PKE-Typ
      SLD   3;
      +AR2;	// Addiere AKKU 1 zum Adreßregister 2
NETWORK
TITLE = Eingestellten Wert IR auswerten und ausgeben
      L     #IR_2;	// Eingestellten IR-Wert laden
      L     0;	// Wert für möglichen Einstellwert laden
      ==I;	// Vergleich
      JNB   _001;	// Sprung wenn nicht gleich
      L     DBD [AR2,P#0.0];	// Wenn Vergleich poistiv dann Wert vom DB holen
      T     #IR_Wert;	// Eingestellten Wert merken
_001: L     #IR_2;
      L     1;
      ==I;
      JNB   _002;
      L     DBD [AR2,P#4.0];
      T     #IR_Wert;
_002: L     #IR_2;
      L     2;
      ==I;
      JNB   _003;
      L     DBD [AR2,P#8.0];
      T     #IR_Wert;
_003: L     #IR_2;
      L     3;
      ==I;
      JNB   _004;
      L     DBD [AR2,P#12.0];
      T     #IR_Wert;
_004: L     #IR_2;
      L     4;
      ==I;
      JNB   _005;
      L     DBD [AR2,P#16.0];
      T     #IR_Wert;
_005: L     #IR_2;
      L     5;
      ==I;
      JNB   _006;
      L     DBD [AR2,P#20.0];
      T     #IR_Wert;
_006: L     #IR_2;
      L     6;
      ==I;
      JNB   _007;
      L     DBD [AR2,P#24.0];
      T     #IR_Wert;
_007: L     #IR_2;
      L     7;
      ==I;
      JNB   _008;
      L     DBD [AR2,P#28.0];
      T     #IR_Wert;
_008: L     #IR_2;
      L     8;
      ==I;
      JNB   _009;
      L     DBD [AR2,P#32.0];
      T     #IR_Wert;
_009: L     #IR_2;
      L     9;
      ==I;
      JNB   _00a;
      L     DBD [AR2,P#36.0];
      T     #IR_Wert;
_00a: L     #IR_2;
      L     10;
      ==I;
      JNB   _00b;
      L     DBD [AR2,P#40.0];
      T     #IR_Wert;
_00b: L     #IR_2;
      L     11;
      ==I;
      JNB   _00c;
      L     DBD [AR2,P#44.0];
      T     #IR_Wert;
_00c: L     #IR_2;
      L     12;
      ==I;
      JNB   _00d;
      L     DBD [AR2,P#48.0];
      T     #IR_Wert;
_00d: L     #IR_2;
      L     13;
      ==I;
      JNB   _00e;
      L     DBD [AR2,P#52.0];
      T     #IR_Wert;
_00e: L     #IR_2;
      L     14;
      ==I;
      JNB   _00f;
      L     DBD [AR2,P#56.0];
      T     #IR_Wert;
_00f: L     #IR_2;
      L     15;
      ==I;
      JNB   _010;
      L     DBD [AR2,P#60.0];
      T     #IR_Wert;
_010: NOP   0;
NETWORK
TITLE = Grenzen für IR-Strom überprüfen
      L     #IR_Strom;	// Eingestellter Stromwert vom PKE
      L     1.050000e+00;	// +5% für Obergrenze
      *R;
      T     #IR_High;	// Merken als oberen Einstellwert
      L     #IR_Wert;	// Eingestellten Wert laden
      L     #IR_High;	// Obergrenze laden
      <=R;	// Vergleich
      =     #Release;	// Eingestellter Wert kleiner als Obergrenze -> Freigabe
NETWORK
TITLE = Wert in DB schreiben
      L     #Daten_DB;	// Nummer des DB laden
      T     #iDBNr;	// Nummer für Instanz DB übertragen
      OPN   DB [#iDBNr];	// Instanz DB öffnen
      LAR1  P#DBX 0.0;	// Lade Adreßregister 1
      L     #Offset;	// Offset für PKE im Datenbaustein
      SLD   3;
      +AR1;	// Addiere AKKU 1 zum Adreßregister 1
      L     #Motorstrom_In;	// Motorstrom laden
      T     DBW [AR1,P#0.0];	// in DB ablegen
      L     #Therm_In;	// Thermischen Motorabbild laden
      T     DBW [AR1,P#2.0];	// in DB ablegen
      L     #IR_Wert;	// Eingestellten IR-Wert laden
      T     DBD [AR1,P#4.0];	// in DB ablegen
      L     #TRIPR_2;	// Auslösegrund laden
      T     DBW [AR1,P#8.0];	// in DB ablegen
      A     #Contactor_In;	// Schaltzustand Schütz laden
      =     DBX [AR1,P#10.0];	// in DB ablegen
      A     #Status_In;	// Status PKE laden
      =     DBX [AR1,P#10.1];	// in DB ablegen
      A     #S_A;	// 1-0-A-Schalter Stellung "A"
      =     DBX [AR1,P#10.2];	// in DB ablegen
      A     #S_0;	// 1-0-A-Schalter Stellung "0"
      =     DBX [AR1,P#10.3];	// in DB ablegen
      A     #S_1;	// 1-0-A-Schalter Stellung "1"
      =     DBX [AR1,P#10.4];	// in DB ablegen
      A     #Failure_In;	// Status Diagnosemeldung laden
      =     DBX [AR1,P#10.5];	// in DB ablegen
      A     #Present_In;	// Status Modul vorhanden laden
      =     DBX [AR1,P#10.6];	// in DB ablegen
      A     #Release;	// Freigabestatus für Einstellstrom laden
      =     DBX [AR1,P#10.7];	// in DB ablegen
END_FUNCTION

FUNCTION "PKE65" : BOOL	// FC 111
TITLE = Motorstarterkombinationen mit PKE
AUTHOR : Simdon
FAMILY : PKE
NAME : PKE-1
VERSION : 0.1
VAR_INPUT
  Daten_DB : INT ;	//Bausteinnummer für Datenablage
  PKE_DB : INT ;	//Bausteinnummer für PKE-Daten
  Offset : INT ;	//Bausteinoffset für Datenablage
  Eingang : INT ;	//Eingangsadresse des PKE (Anfangsadresse)
  IR_Strom : REAL ;	//Maximaler Einstellwert für PKE
END_VAR
VAR_OUTPUT
  RET_VAL : BOOL ;
END_VAR
VAR_TEMP
  Contactor_In : BOOL ;	//Schaltstellung Leistungsschütz
  Status_In : BOOL ;	//Status PKE
  Auto_In : BOOL ;	//Stellung Schalter 1-0-A
  Auto2_In : BOOL ;	//Stellung Schalter 1-0-A
  Failure_In : BOOL ;	//Diagnosemeldung
  Frei1_In : BOOL ;
  Present_In : BOOL ;	//Modul vorhanden
  Frei2_In : BOOL ;
  IR1_In : BOOL ;	//Eingestellter Wert IR
  IR2_In : BOOL ;	//Eingestellter Wert IR
  IR3_In : BOOL ;	//Eingestellter Wert IR
  IR4_In : BOOL ;	//Eingestellter Wert IR
  TRIPR1_In : BOOL ;	//Auslösegrund
  TRIPR2_In : BOOL ;	//Auslösegrund
  TRIPR3_In : BOOL ;	//Auslösegrund
  ACKR_In : BOOL ;	//Acknowledge
  Motorstrom_In : BYTE ;	//Motorstrom
  Therm_In : BYTE ;	//Thermisches Motorabbild
  Block_In : BYTE ;	//Auslöseblock
  IR_1 : WORD ;	//Zwischenwert Auslösestrom
  IR_2 : INT ;	//Zwischenwert Auslösestrom
  TRIPR_1 : WORD ;	//Zwischenwert Auslösegrund
  TRIPR_2 : INT ;	//Zwischenwert Auslösegrund
  IR_Wert : REAL ;	//Gewandelter Wert für Auslösestrom
  IR_High : REAL ;	//Obergrenze für Auslösestrom
  Release : BOOL ;	//Freigabe wenn eingestellter Auslösestrom okay
  iDBNr : INT ;	//Instanz-DB für Datenablage
  Offset2 : INT ;	//Offset für PKE-DB
  EAAdr : DINT ;	//Eingangsadresse für PKE
  RetVal : INT ;
  Block1 : WORD ;	//Zwischenwert für Typ Auslöseblock
  Block2 : INT ;	//Zwischenwert für Typ Auslöseblock
  S_A : BOOL ;	//Stellung 1-0-A-Schalter "A"
  S_0 : BOOL ;	//Stellung 1-0-A-Schalter "0"
  S_1 : BOOL ;	//Stellung 1-0-A-Schalter "1"
  iDB_PKE : INT ;	//Instanz-DB für PKE-Daten
END_VAR
BEGIN
NETWORK
TITLE = Eingangswerte laden und verteilen
      L     #Eingang;	// Anfangsadresse des PKE
      T     #EAAdr;	// Übertragen in temp. Adressmerker
      SLD   3;	// Wort schieben
      LAR1;	// Wert ins Adressregister 1 ablegen
      L     PIB [AR1,P#0.0];	// Eingangsbyte laden
      T     LB 0;	// In Lokaldaten ablegen
      L     PIB [AR1,P#1.0];	// Eingangsbyte laden
      T     LB 1;	// In Lokaldaten ablegen
      L     PIB [AR1,P#2.0];	// Eingangsbyte laden
      T     #Motorstrom_In;	// In Lokaldaten ablegen
      L     PIB [AR1,P#3.0];	// Eingangsbyte laden
      T     #Therm_In;	// In Lokaldaten ablegen
      L     PIB [AR1,P#4.0];	// Eingangsbyte laden
      T     #Block_In;	// In Lokaldaten ablegen
NETWORK
TITLE = Feststellen welcher Auslöseblock eingesetzt wird
      L     #Block_In;	// Kenndaten vom Auslöseblock lesen
      T     #Block1;	// Wandlung zum Wort
      L     W#16#7;	// Typ Auslöseblock maskieren
      AW;
      T     #Block2;	// Als Integer ablegen
      L     #Block2;	// Blocktyp laden
      L     0;	// Vergleich mit PKE 1,2
      ==I;
      JNB   _011;	// Sprung wenn nicht gleich
      L     0;	// Offset für DB zum Datenauslesen
      T     #Offset2;
_011: L     #Block2;	// Blocktyp laden
      L     1;	// Vergleich mit PKE 4
      ==I;
      JNB   _012;	// Sprung wenn nicht gleich
      L     64;	// Offset für DB zum Datenauslesen
      T     #Offset2;	// Offset ablegen
_012: L     #Block2;	// Blocktyp laden
      L     2;	// Vergleich mit PKE 12
      ==I;
      JNB   _013;	// Sprung wenn nicht gleich
      L     128;	// Offset für DB zum Datenauslesen
      T     #Offset2;	// Offset ablegen
_013: L     #Block2;	// Blocktyp laden
      L     3;	// Vergleich mit PKE 32
      ==I;
      JNB   _014;	// Sprung wenn nicht gleich
      L     192;	// Offset für DB zum Datenauslesen
      T     #Offset2;	// Offset ablegen
_014: L     #Block2;	// Blocktyp laden
      L     5;	// Vergleich mit PKE 65
      ==I;
      JNB   _015;	// Sprung wenn nicht gleich
      L     256;	// Offset für DB zum Datenauslesen
      T     #Offset2;	// Offset ablegen
_015: NOP   0;
NETWORK
TITLE = Eingestellten Wert IR maskieren und wandeln
      L     LB 1;	// Byte 1 vom PKE laden
      T     #IR_1;	// Zwischenspeichern in IR-Werte 1
      L     W#16#F;	// Eingestellten IR-Wert maskieren
      AW;
      T     #IR_2;	// IR-Wert als Integer
NETWORK
TITLE = Auslösegrung TRIPR maskieren und wandeln
//1: Überlastfall; 2: Kurzschluß; 3: Phasenausfall/Phasenunsymetrie
//4: Stellung Test am PKE
      L     LB 1;	// Byte 1 vom PKE laden
      L     #TRIPR_1;	// Zwischenspeichern in TRIPR-Werte 1
      L     W#16#70;	// TRIPR-Wert maskieren
      AW;
      T     #TRIPR_2;	// TRIPR-Wert als Integer
NETWORK
TITLE = Auswertung 1-0-A-Schalter
      A     #Auto_In;	// Stellung 1-0-A-Schalter Bit 1
      AN    #Auto2_In;	// Stellung 1-0-A-Schalter Bit 2
      =     #S_A;	// Schalter in Stellung "A"
      AN    #Auto_In;	// Stellung 1-0-A-Schalter Bit 1
      A     #Auto2_In;	// Stellung 1-0-A-Schalter Bit 2
      =     #S_0;	// Schalter in Stellung "0"
      A     #Auto_In;	// Stellung 1-0-A-Schalter Bit 1
      A     #Auto2_In;	// Stellung 1-0-A-Schalter Bit 2
      =     #S_1;	// Schalter in Stellung "1"
NETWORK
TITLE = DB mit IR Werten für PKE öffnen
      L     #PKE_DB;	// Nummer des DB laden
      T     #iDB_PKE;	// Nummer für Instanz DB übertragen
      OPN   DB [#iDB_PKE];	// Instanz DB öffnen
      LAR2  P#DBX 0.0;	// Pointer auf Anfang
      L     #Offset2;	// Offset für PKE-Typ
      SLD   3;
      +AR2;	// Addiere AKKU 1 zum Adreßregister 2
NETWORK
TITLE = Eingestellten Wert IR auswerten und ausgeben
      L     #IR_2;	// Eingestellten IR-Wert laden
      L     0;	// Wert für möglichen Einstellwert laden
      ==I;	// Vergleich
      JNB   _001;	// Sprung wenn nicht gleich
      L     DBD [AR2,P#0.0];	// Wenn Vergleich poistiv dann Wert vom DB holen
      T     #IR_Wert;	// Eingestellten Wert merken
_001: L     #IR_2;
      L     1;
      ==I;
      JNB   _002;
      L     DBD [AR2,P#4.0];
      T     #IR_Wert;
_002: L     #IR_2;
      L     2;
      ==I;
      JNB   _003;
      L     DBD [AR2,P#8.0];
      T     #IR_Wert;
_003: L     #IR_2;
      L     3;
      ==I;
      JNB   _004;
      L     DBD [AR2,P#12.0];
      T     #IR_Wert;
_004: L     #IR_2;
      L     4;
      ==I;
      JNB   _005;
      L     DBD [AR2,P#16.0];
      T     #IR_Wert;
_005: L     #IR_2;
      L     5;
      ==I;
      JNB   _006;
      L     DBD [AR2,P#20.0];
      T     #IR_Wert;
_006: L     #IR_2;
      L     6;
      ==I;
      JNB   _007;
      L     DBD [AR2,P#24.0];
      T     #IR_Wert;
_007: L     #IR_2;
      L     7;
      ==I;
      JNB   _008;
      L     DBD [AR2,P#28.0];
      T     #IR_Wert;
_008: L     #IR_2;
      L     8;
      ==I;
      JNB   _009;
      L     DBD [AR2,P#32.0];
      T     #IR_Wert;
_009: L     #IR_2;
      L     9;
      ==I;
      JNB   _00a;
      L     DBD [AR2,P#36.0];
      T     #IR_Wert;
_00a: L     #IR_2;
      L     10;
      ==I;
      JNB   _00b;
      L     DBD [AR2,P#40.0];
      T     #IR_Wert;
_00b: L     #IR_2;
      L     11;
      ==I;
      JNB   _00c;
      L     DBD [AR2,P#44.0];
      T     #IR_Wert;
_00c: L     #IR_2;
      L     12;
      ==I;
      JNB   _00d;
      L     DBD [AR2,P#48.0];
      T     #IR_Wert;
_00d: L     #IR_2;
      L     13;
      ==I;
      JNB   _00e;
      L     DBD [AR2,P#52.0];
      T     #IR_Wert;
_00e: L     #IR_2;
      L     14;
      ==I;
      JNB   _00f;
      L     DBD [AR2,P#56.0];
      T     #IR_Wert;
_00f: L     #IR_2;
      L     15;
      ==I;
      JNB   _010;
      L     DBD [AR2,P#60.0];
      T     #IR_Wert;
_010: NOP   0;
NETWORK
TITLE = Grenzen für IR-Strom überprüfen
      L     #IR_Strom;	// Eingestellter Stromwert vom PKE
      L     1.050000e+00;	// +5% für Obergrenze
      *R;
      T     #IR_High;	// Merken als oberen Einstellwert
      L     #IR_Wert;	// Eingestellten Wert laden
      L     #IR_High;	// Obergrenze laden
      <=R;	// Vergleich
      =     #Release;	// Eingestellter Wert kleiner als Obergrenze -> Freigabe
NETWORK
TITLE = Wert in DB schreiben
      L     #Daten_DB;	// Nummer des DB laden
      T     #iDBNr;	// Nummer für Instanz DB übertragen
      OPN   DB [#iDBNr];	// Instanz DB öffnen
      LAR1  P#DBX 0.0;	// Lade Adreßregister 1
      L     #Offset;	// Offset für PKE im Datenbaustein
      SLD   3;
      +AR1;	// Addiere AKKU 1 zum Adreßregister 1
      L     #Motorstrom_In;	// Motorstrom laden
      T     DBW [AR1,P#0.0];	// in DB ablegen
      L     #Therm_In;	// Thermischen Motorabbild laden
      T     DBW [AR1,P#2.0];	// in DB ablegen
      L     #IR_Wert;	// Eingestellten IR-Wert laden
      T     DBD [AR1,P#4.0];	// in DB ablegen
      L     #TRIPR_2;	// Auslösegrund laden
      T     DBW [AR1,P#8.0];	// in DB ablegen
      A     #Contactor_In;	// Schaltzustand Schütz laden
      =     DBX [AR1,P#10.0];	// in DB ablegen
      A     #Status_In;	// Status PKE laden
      =     DBX [AR1,P#10.1];	// in DB ablegen
      A     #S_A;	// 1-0-A-Schalter Stellung "A"
      =     DBX [AR1,P#10.2];	// in DB ablegen
      A     #S_0;	// 1-0-A-Schalter Stellung "0"
      =     DBX [AR1,P#10.3];	// in DB ablegen
      A     #S_1;	// 1-0-A-Schalter Stellung "1"
      =     DBX [AR1,P#10.4];	// in DB ablegen
      A     #Failure_In;	// Status Diagnosemeldung laden
      =     DBX [AR1,P#10.5];	// in DB ablegen
      A     #Present_In;	// Status Modul vorhanden laden
      =     DBX [AR1,P#10.6];	// in DB ablegen
      A     #Release;	// Freigabestatus für Einstellstrom laden
      =     DBX [AR1,P#10.7];	// in DB ablegen
END_FUNCTION

FUNCTION "AltivarControl" : VOID	// FC 112
TITLE = Profibusanbindung für Schneider Altivar
AUTHOR : Simdon
FAMILY : Motoren
NAME : Altivar
VERSION : 0.1
VAR_INPUT
  DB_Nr : INT ;	//Datenbausteinnummer
  Offset : INT ;	//Offsetwert für den Umrichter
  Anz_PZD : INT ;	//Anzahl der PZD-Worte vom Umrichter
  DrehzahlSoll : WORD ;	//Drehzahl Sollwert
  Ein_Aus : BOOL ;	//Ein-Aus Befehl
  Stoer_Quit : BOOL ;	//Störung Quittieren
END_VAR
VAR_OUTPUT
  RPMOut : INT ;
  BetrStd : INT ;
  MotorSpg : INT ;
  NetzSpg : INT ;
  MotorLstg : INT ;
  Motorstrom : INT ;
  Fehlercode : INT ;
  Busfehler : BOOL ;
  InBetrieb : BOOL ;
  Stoerung : BOOL ;
  Alarm : BOOL ;
END_VAR
VAR_TEMP
  iDBNr : INT ;	//Instanzdatenbaustein
  StartNr : INT ;	//Adresse des ersten PEW
  PEWco : INT ;	//Counter für PEW
  AnzLoop : INT ;	//Anzahl der zu lesenden Worte
  LDco : INT ;	//Counter für Lokaldaten-Ablage
  PZDAus_1 : WORD ;	//PZD-Statuswort Altivar
  PZDAus_2 : WORD ;	//PZD-Ausgangswort 2
  PZDAus_3 : WORD ;	//PZD-Ausgangswort 3
  PZDAus_4 : WORD ;	//PZD-Ausgangswort 4
  PZDAus_5 : WORD ;	//PZD-Ausgangswort 5
  PZDAus_6 : WORD ;	//PZD-Ausgangswort 6
  PZDAus_7 : WORD ;	//PZD-Ausgangswort 7
  PZDAus_8 : WORD ;	//PZD-Ausgangswort 8
  RetVal : INT ;
  EAadr : WORD ;
END_VAR
BEGIN
NETWORK
TITLE = Datenbaustein öffnen und Startadresse für erstes PEW setzen
      L     #DB_Nr;	// Nummer des DB laden
      T     #iDBNr;	// Nummer für Instanz DB übertragen
      OPN   DB [#iDBNr];	// Instanz DB öffnen
      LAR1  P#DBX 0.0;
      L     #Offset;
      SLD   3;
      +AR1;
      L     DBW [AR1,P#0.0];	// Erstes Datenwort lesen
      T     #StartNr;	// Merken des ersten PEW
NETWORK
TITLE = Daten vom Umrichter lesen (8 Worte aus dem PZD-Bereich)
      L     10;	// Ausgabeadresse für 1.PEW laden  (PZD Statuswort Altivar)
      T     #LDco;	// Merken der Ausgabeadresse für 1.PEW (Lokaldatenspeicher)
      SLW   3;	// Umwandeln ins Pointerformat
      LAR2;	// Adressregister 2 laden
      L     0;	// Zähler für PEW initialisieren
      T     #PEWco;	// Merken des Zählers für die PEW
      L     #Anz_PZD;	// Anzahl der Schleifendurchläufe laden
next: T     #AnzLoop;	// Schleife starten
      L     #StartNr;	// Adresse des 1.PEW laden
      L     #PEWco;	// Schrittweite für die PEW laden
      +I;	// Zur vorherigen PEW-Adresse addieren
      SLW   3;	// Umwandlung des aktuellen PEW in das Pointerformat
      LAR1;	// Adressregister 1 laden
      L     PIW [AR1,P#0.0];	// PEW mit Adresse aus ADR1 lesen
      T     LW [AR2,P#0.0];	// Speichern des aktuellen PEW im Lokaldatenspeicher
      L     #PEWco;	// Adresse des aktuellen PEW laden
      L     2;	// Schrittweite für PEW laden
      +I;	// Beides addieren
      T     #PEWco;	// Neues PEW merken
      L     #LDco;	// Aktuelle Ausgabeadresse laden
      L     2;	// Schrittweite für Ausgabe-PEW laden
      +I;	// Beides addieren
      T     #LDco;	// Merken des neuen Ausgabe-PEW
      SLW   3;	// Umwandeln ins Pointerformat
      LAR2;	// Adressregister 2 laden
      L     #AnzLoop;	// Schleifenzähler -1
      LOOP  next;	// Ende der Schleife
NETWORK
TITLE = Ausgabedaten des Umrichters im DB speichern (nicht skaliert)
      LAR1  P#DBX 0.0;	// Startadresse aus dem DB lesen
      L     #Offset;	// Offset laden
      SLD   3;	// Umwandeln ins Pointerformat
      +AR1;	// Im Adressregister 1 ablegen
      L     #PZDAus_1;	// Statuswort laden
      T     DBW [AR1,P#22.0];
      A     DBX [AR1,P#22.1];
      =     #Busfehler;
      A     DBX [AR1,P#23.2];
      =     #InBetrieb;
      A     DBX [AR1,P#23.3];
      =     #Stoerung;
      A     DBX [AR1,P#23.7];
      =     #Alarm;
      L     #PZDAus_2;	// Drehzahl in U/min
      T     DBW [AR1,P#24.0];
      T     #RPMOut;
      L     #PZDAus_3;	// Betriebsstunden Motor
      T     DBW [AR1,P#26.0];
      T     #BetrStd;
      L     #PZDAus_4;	// Motorspannung in 1 Volt
      T     DBW [AR1,P#28.0];
      T     #MotorSpg;
      L     #PZDAus_5;	// Netzspannung in 0,1 Volt
      L     10;
      *I;
      T     DBW [AR1,P#30.0];
      T     #NetzSpg;
      L     #PZDAus_6;	// Motorleistung in 1 Prozent
      T     DBW [AR1,P#32.0];
      T     #MotorLstg;
      L     #PZDAus_7;	// Motornennstrom in 0,1 Ampere
      L     10;
      *I;
      T     DBW [AR1,P#34.0];
      T     #Motorstrom;
      L     #PZDAus_8;	// Altivar Fehlercode
      T     DBW [AR1,P#36.0];
      T     #Fehlercode;
NETWORK
TITLE = FU CMD Steuerwort Freigabe Spannung, Schnellhalt Ein
      A     DBX [AR1,P#22.1];	// Bus-Fehler
      AN    DBX [AR1,P#23.3];	// FU Störung
      =     DBX [AR1,P#3.2];	// Schnellhalt
      =     DBX [AR1,P#3.1];	// Freigabe Spannung
NETWORK
TITLE = Störung Quittieren
      A     #Stoer_Quit;
      =     DBX [AR1,P#3.7];	// Stoerung Quittieren
NETWORK
TITLE = FU CMD Steuerwort  FU - Einschaltung u. Freigabe Betrieb
      A     #Ein_Aus;
      S     DBX [AR1,P#3.0];	// FU Einschalten
      A(;
      ON    DBX [AR1,P#3.1];	// Freigabe Spannung
      ON    DBX [AR1,P#3.2];	// Schnellhalt
      ON    #Ein_Aus;
      );
      R     DBX [AR1,P#3.0];	// FU Einschalten
      A     DBX [AR1,P#3.0];	// FU Einschalten
      =     DBX [AR1,P#3.3];	// Freigabe Betrieb
NETWORK
TITLE = Daten zum Umrichter: CMD-Wort u. Drehzahlsollwert
      L     #StartNr;
      SLW   3;
      LAR2;
      L     DBW [AR1,P#2.0];	// CMD-Wort lesen
      T     PQW [AR2,P#0.0];	// CMD-Wort zum Umrichter senden
      L     #DrehzahlSoll;	// Drehzahlsollwert lesen
      T     PQW [AR2,P#2.0];	// Drehzahlsollwert zum Umrichter ausgeben
END_FUNCTION

// FC 125: know-how protected block, not included

FUNCTION "SYS_DT" : VOID	// FC 126
TITLE = Systemzeit
AUTHOR : Simdon
NAME : SYS_DT
VERSION : 0.1
VAR_TEMP
  DT1 : DATE_AND_TIME ;
  DT2 : DATE_AND_TIME ;
  DT3 : DATE_AND_TIME ;
  Zahl1 : DINT ;
  Zahl2 : DINT ;
  Zahl3 : TIME ;
  Zahl4 : INT ;
  J1 : INT ;
  J1_BCD : WORD ;
  M1_BCD : WORD ;
  T1_BCD : WORD ;
END_VAR
BEGIN
